  MoveL 6726 to (240.81, 149.3, 97.46) mm, rotated rx -180 ry 0 rz 180 deg; joints [-61.575, 61.202, -81.531, 63.09, 99.519, 18.047]
  Call Extruder(259.46531)
  MoveL 6727 to (240.76, 149.6, 97.46) mm, rotated rx 180 ry 0 rz 180 deg; joints [-61.639, 61.223, -81.522, 63.147, 99.485, 18.03]
  MoveL 6728 to (240.76, 149.6, 97.46) mm, rotated rx 180 ry 0 rz 180 deg; joints [-61.639, 61.223, -81.522, 63.147, 99.485, 18.03]
  Call Extruder(259.62559)
  MoveL 6729 to (240.71, 149.91, 97.46) mm, rotated rx -180 ry 0 rz -180 deg; joints [-61.702, 61.244, -81.513, 63.203, 99.453, 18.013]
  MoveL 6730 to (240.71, 149.91, 97.46) mm, rotated rx -180 ry 0 rz -180 deg; joints [-61.702, 61.244, -81.513, 63.203, 99.453, 18.013]
  Call Extruder(259.78661)
  MoveL 6731 to (240.66, 150.21, 97.46) mm, rotated rx -180 ry 0 rz -180 deg; joints [-61.765, 61.265, -81.504, 63.26, 99.419, 17.996]
  MoveL 6732 to (240.66, 150.21, 97.46) mm, rotated rx -180 ry 0 rz -180 deg; joints [-61.765, 61.265, -81.504, 63.26, 99.419, 17.996]
  Call Extruder(259.94835)
  MoveL 6733 to (240.61, 150.52, 97.46) mm, rotated rx 180 ry 0 rz 180 deg; joints [-61.828, 61.286, -81.495, 63.316, 99.387, 17.979]
  MoveL 6734 to (240.61, 150.52, 97.46) mm, rotated rx 180 ry 0 rz 180 deg; joints [-61.828, 61.286, -81.495, 63.316, 99.387, 17.979]
  Call Extruder(260.11082)
  MoveL 6735 to (240.56, 150.83, 97.46) mm, rotated rx 180 ry 0 rz 180 deg; joints [-61.891, 61.307, -81.486, 63.372, 99.354, 17.961]
  MoveL 6736 to (240.56, 150.83, 97.46) mm, rotated rx 180 ry 0 rz 180 deg; joints [-61.891, 61.307, -81.486, 63.372, 99.354, 17.961]
  Call Extruder(260.24475)
  MoveL 6737 to (240.52, 151.08, 97.46) mm, rotated rx -180 ry 0 rz 180 deg; joints [-61.944, 61.324, -81.479, 63.42, 99.327, 17.948]
  MoveL 6738 to (240.52, 151.08, 97.46) mm, rotated rx -180 ry 0 rz 180 deg; joints [-61.944, 61.324, -81.479, 63.42, 99.327, 17.948]
  Call Extruder(260.37929)
  MoveL 6739 to (240.47, 151.32, 97.46) mm, rotated rx -180 ry 0 rz 180 deg; joints [-61.998, 61.34, -81.472, 63.469, 99.299, 17.935]
  MoveL 6740 to (240.47, 151.32, 97.46) mm, rotated rx -180 ry 0 rz 180 deg; joints [-61.998, 61.34, -81.472, 63.469, 99.299, 17.935]
  Call Extruder(260.51443)
  MoveL 6741 to (240.42, 151.57, 97.46) mm, rotated rx -180 ry 0 rz 180 deg; joints [-62.052, 61.357, -81.465, 63.517, 99.272, 17.922]
  MoveL 6742 to (240.42, 151.57, 97.46) mm, rotated rx -180 ry 0 rz 180 deg; joints [-62.052, 61.357, -81.465, 63.517, 99.272, 17.922]
  Call Extruder(260.65019)
  MoveL 6743 to (240.37, 151.82, 97.46) mm, rotated rx 180 ry 0 rz -180 deg; joints [-62.105, 61.374, -81.458, 63.565, 99.245, 17.908]
  MoveL 6744 to (240.37, 151.82, 97.46) mm, rotated rx 180 ry 0 rz -180 deg; joints [-62.105, 61.374, -81.458, 63.565, 99.245, 17.908]
  Call Extruder(260.78656)
  MoveL 6745 to (240.32, 152.07, 97.46) mm, rotated rx 180 ry 0 rz -180 deg; joints [-62.159, 61.39, -81.45, 63.613, 99.218, 17.895]
  MoveL 6746 to (240.32, 152.07, 97.46) mm, rotated rx 180 ry 0 rz -180 deg; joints [-62.159, 61.39, -81.45, 63.613, 99.218, 17.895]
  Call Extruder(260.92354)
  MoveL 6747 to (240.27, 152.32, 97.46) mm, rotated rx -180 ry 0 rz 180 deg; joints [-62.212, 61.407, -81.443, 63.661, 99.191, 17.881]
  MoveL 6748 to (240.27, 152.32, 97.46) mm, rotated rx -180 ry 0 rz 180 deg; joints [-62.212, 61.407, -81.443, 63.661, 99.191, 17.881]
  Call Extruder(261.06113)
  MoveL 6749 to (240.22, 152.57, 97.46) mm, rotated rx -180 ry 0 rz 180 deg; joints [-62.265, 61.424, -81.436, 63.709, 99.164, 17.868]
  MoveL 6750 to (240.22, 152.57, 97.46) mm, rotated rx -180 ry 0 rz 180 deg; joints [-62.265, 61.424, -81.436, 63.709, 99.164, 17.868]
  Call Extruder(261.17482)
  MoveL 6751 to (240.17, 152.77, 97.46) mm, rotated rx -180 ry 0 rz 180 deg; joints [-62.31, 61.437, -81.43, 63.749, 99.142, 17.857]
  MoveL 6752 to (240.17, 152.77, 97.46) mm, rotated rx -180 ry 0 rz 180 deg; joints [-62.31, 61.437, -81.43, 63.749, 99.142, 17.857]
  Call Extruder(261.28897)
  MoveL 6753 to (240.13, 152.98, 97.46) mm, rotated rx 180 ry 0 rz 180 deg; joints [-62.355, 61.451, -81.424, 63.789, 99.119, 17.846]
  MoveL 6754 to (240.13, 152.98, 97.46) mm, rotated rx 180 ry 0 rz 180 deg; joints [-62.355, 61.451, -81.424, 63.789, 99.119, 17.846]
  Call Extruder(261.40358)
  MoveL 6755 to (240.08, 153.18, 97.46) mm, rotated rx -180 ry 0 rz 180 deg; joints [-62.399, 61.464, -81.418, 63.83, 99.097, 17.835]
  MoveL 6756 to (240.08, 153.18, 97.46) mm, rotated rx -180 ry 0 rz 180 deg; joints [-62.399, 61.464, -81.418, 63.83, 99.097, 17.835]
  Call Extruder(261.51863)
  MoveL 6757 to (240.04, 153.39, 97.46) mm, rotated rx -180 ry 0 rz 180 deg; joints [-62.444, 61.478, -81.412, 63.869, 99.075, 17.824]
  MoveL 6758 to (240.04, 153.39, 97.46) mm, rotated rx -180 ry 0 rz 180 deg; joints [-62.444, 61.478, -81.412, 63.869, 99.075, 17.824]
  Call Extruder(261.64086)
  MoveL 6759 to (239.98, 153.6, 97.46) mm, rotated rx -180 ry 0 rz -180 deg; joints [-62.493, 61.492, -81.406, 63.914, 99.051, 17.813]
  MoveL 6760 to (239.98, 153.6, 97.46) mm, rotated rx -180 ry 0 rz -180 deg; joints [-62.493, 61.492, -81.406, 63.914, 99.051, 17.813]
  Call Extruder(261.77052)
  MoveL 6761 to (239.92, 153.82, 97.46) mm, rotated rx -180 ry 0 rz 180 deg; joints [-62.547, 61.506, -81.4, 63.963, 99.026, 17.803]
  MoveL 6762 to (239.92, 153.82, 97.46) mm, rotated rx -180 ry 0 rz 180 deg; joints [-62.547, 61.506, -81.4, 63.963, 99.026, 17.803]
  Call Extruder(261.90074)
  MoveL 6763 to (239.85, 154.05, 97.46) mm, rotated rx 180 ry 0 rz 180 deg; joints [-62.601, 61.52, -81.394, 64.012, 99, 17.793]
  MoveL 6764 to (239.85, 154.05, 97.46) mm, rotated rx 180 ry 0 rz 180 deg; joints [-62.601, 61.52, -81.394, 64.012, 99, 17.793]
  Call Extruder(262.03153)
  MoveL 6765 to (239.78, 154.27, 97.46) mm, rotated rx -180 ry 0 rz -180 deg; joints [-62.654, 61.534, -81.387, 64.061, 98.975, 17.782]
  MoveL 6766 to (239.78, 154.27, 97.46) mm, rotated rx -180 ry 0 rz -180 deg; joints [-62.654, 61.534, -81.387, 64.061, 98.975, 17.782]
  Call Extruder(262.16289)
  MoveL 6767 to (239.71, 154.49, 97.46) mm, rotated rx -180 ry 0 rz 180 deg; joints [-62.708, 61.548, -81.381, 64.11, 98.95, 17.772]
  MoveL 6768 to (239.71, 154.49, 97.46) mm, rotated rx -180 ry 0 rz 180 deg; joints [-62.708, 61.548, -81.381, 64.11, 98.95, 17.772]
  Call Extruder(262.27479)
  MoveL 6769 to (239.65, 154.68, 97.46) mm, rotated rx -180 ry 0 rz 180 deg; joints [-62.754, 61.56, -81.376, 64.152, 98.928, 17.763]
  MoveL 6770 to (239.65, 154.68, 97.46) mm, rotated rx -180 ry 0 rz 180 deg; joints [-62.754, 61.56, -81.376, 64.152, 98.928, 17.763]
  Call Extruder(262.38714)
  MoveL 6771 to (239.59, 154.87, 97.46) mm, rotated rx -180 ry 0 rz 180 deg; joints [-62.801, 61.572, -81.371, 64.195, 98.907, 17.754]
  MoveL 6772 to (239.59, 154.87, 97.46) mm, rotated rx -180 ry 0 rz 180 deg; joints [-62.801, 61.572, -81.371, 64.195, 98.907, 17.754]
  Call Extruder(262.49993)
  MoveL 6773 to (239.53, 155.06, 97.46) mm, rotated rx -180 ry 0 rz 180 deg; joints [-62.847, 61.584, -81.365, 64.237, 98.885, 17.746]
  MoveL 6774 to (239.53, 155.06, 97.46) mm, rotated rx -180 ry 0 rz 180 deg; joints [-62.847, 61.584, -81.365, 64.237, 98.885, 17.746]
  Call Extruder(262.61316)
  MoveL 6775 to (239.47, 155.25, 97.46) mm, rotated rx -180 ry 0 rz 180 deg; joints [-62.893, 61.595, -81.36, 64.279, 98.864, 17.737]
  MoveL 6776 to (239.47, 155.25, 97.46) mm, rotated rx -180 ry 0 rz 180 deg; joints [-62.893, 61.595, -81.36, 64.279, 98.864, 17.737]
  Call Extruder(262.72684)
  MoveL 6777 to (239.41, 155.44, 97.46) mm, rotated rx 180 ry 0 rz -180 deg; joints [-62.939, 61.607, -81.355, 64.321, 98.842, 17.729]
  MoveL 6778 to (239.41, 155.44, 97.46) mm, rotated rx 180 ry 0 rz -180 deg; joints [-62.939, 61.607, -81.355, 64.321, 98.842, 17.729]
  Call Extruder(262.90880)
  MoveL 6779 to (239.29, 155.73, 97.46) mm, rotated rx 180 ry 0 rz 180 deg; joints [-63.018, 61.624, -81.347, 64.393, 98.807, 17.717]
  MoveL 6780 to (239.29, 155.73, 97.46) mm, rotated rx 180 ry 0 rz 180 deg; joints [-63.018, 61.624, -81.347, 64.393, 98.807, 17.717]
  Call Extruder(263.09151)
  MoveL 6781 to (239.17, 156.02, 97.46) mm, rotated rx 180 ry 0 rz 180 deg; joints [-63.097, 61.642, -81.339, 64.466, 98.773, 17.706]
  MoveL 6782 to (239.17, 156.02, 97.46) mm, rotated rx 180 ry 0 rz 180 deg; joints [-63.097, 61.642, -81.339, 64.466, 98.773, 17.706]
  Call Extruder(263.26194)
  MoveL 6783 to (239.05, 156.29, 97.46) mm, rotated rx 180 ry 0 rz -180 deg; joints [-63.17, 61.657, -81.332, 64.533, 98.74, 17.696]
  MoveL 6784 to (239.05, 156.29, 97.46) mm, rotated rx 180 ry 0 rz -180 deg; joints [-63.17, 61.657, -81.332, 64.533, 98.74, 17.696]
  Call Extruder(263.41995)
  MoveL 6785 to (238.94, 156.54, 97.46) mm, rotated rx -180 ry 0 rz -180 deg; joints [-63.238, 61.672, -81.325, 64.596, 98.711, 17.686]
  MoveL 6786 to (238.94, 156.54, 97.46) mm, rotated rx -180 ry 0 rz -180 deg; joints [-63.238, 61.672, -81.325, 64.596, 98.711, 17.686]
  Call Extruder(263.57856)
  MoveL 6787 to (238.84, 156.79, 97.46) mm, rotated rx -180 ry 0 rz -180 deg; joints [-63.306, 61.687, -81.319, 64.658, 98.681, 17.677]
  MoveL 6788 to (238.84, 156.79, 97.46) mm, rotated rx -180 ry 0 rz -180 deg; joints [-63.306, 61.687, -81.319, 64.658, 98.681, 17.677]
  Call Extruder(263.78473)
  MoveL 6789 to (238.66, 157.09, 97.46) mm, rotated rx -180 ry 0 rz 180 deg; joints [-63.401, 61.703, -81.311, 64.747, 98.642, 17.669]
  MoveL 6790 to (238.66, 157.09, 97.46) mm, rotated rx -180 ry 0 rz 180 deg; joints [-63.401, 61.703, -81.311, 64.747, 98.642, 17.669]
  Call Extruder(263.99168)
  MoveL 6791 to (238.49, 157.4, 97.46) mm, rotated rx 180 ry 0 rz 180 deg; joints [-63.497, 61.719, -81.304, 64.836, 98.603, 17.661]
  MoveL 6792 to (238.49, 157.4, 97.46) mm, rotated rx 180 ry 0 rz 180 deg; joints [-63.497, 61.719, -81.304, 64.836, 98.603, 17.661]
  Call Extruder(264.19941)
  MoveL 6793 to (238.31, 157.7, 97.46) mm, rotated rx 180 ry 0 rz 180 deg; joints [-63.592, 61.735, -81.297, 64.924, 98.564, 17.653]
  MoveL 6794 to (238.31, 157.7, 97.46) mm, rotated rx 180 ry 0 rz 180 deg; joints [-63.592, 61.735, -81.297, 64.924, 98.564, 17.653]
  Call Extruder(264.40791)
  MoveL 6795 to (238.13, 158.01, 97.46) mm, rotated rx 180 ry 0 rz 180 deg; joints [-63.687, 61.752, -81.289, 65.013, 98.525, 17.645]
  MoveL 6796 to (238.13, 158.01, 97.46) mm, rotated rx 180 ry 0 rz 180 deg; joints [-63.687, 61.752, -81.289, 65.013, 98.525, 17.645]
  Call Extruder(264.58745)
  MoveL 6797 to (237.96, 158.25, 97.46) mm, rotated rx 180 ry 0 rz 180 deg; joints [-63.774, 61.763, -81.284, 65.094, 98.491, 17.642]
  MoveL 6798 to (237.96, 158.25, 97.46) mm, rotated rx 180 ry 0 rz 180 deg; joints [-63.774, 61.763, -81.284, 65.094, 98.491, 17.642]
  Call Extruder(264.92086)
  MoveL 6799 to (237.63, 158.7, 97.46) mm, rotated rx -180 ry 0 rz -180 deg; joints [-63.934, 61.785, -81.274, 65.244, 98.43, 17.635]
  MoveL 6800 to (237.63, 158.7, 97.46) mm, rotated rx -180 ry 0 rz -180 deg; joints [-63.934, 61.785, -81.274, 65.244, 98.43, 17.635]
  Call Extruder(265.25545)
  MoveL 6801 to (237.3, 159.15, 97.46) mm, rotated rx 180 ry 0 rz 180 deg; joints [-64.094, 61.807, -81.263, 65.393, 98.368, 17.628]
  Call Extruder(266.08341)
  MoveL 6802 to (236.39, 160.19, 97.46) mm, rotated rx -180 ry 0 rz -180 deg; joints [-64.505, 61.852, -81.243, 65.781, 98.216, 17.625]
  Call Extruder(266.91134)
  MoveL 6803 to (235.35, 161.1, 97.46) mm, rotated rx 180 ry 0 rz -180 deg; joints [-64.933, 61.884, -81.228, 66.187, 98.068, 17.64]
  Call Extruder(267.07865)
  MoveL 6804 to (235.13, 161.27, 97.46) mm, rotated rx -180 ry 0 rz 180 deg; joints [-65.021, 61.888, -81.226, 66.271, 98.038, 17.646]
  MoveL 6805 to (235.13, 161.27, 97.46) mm, rotated rx -180 ry 0 rz 180 deg; joints [-65.021, 61.888, -81.226, 66.271, 98.038, 17.646]
  Call Extruder(267.41207)
  MoveL 6806 to (234.68, 161.6, 97.46) mm, rotated rx 180 ry 0 rz 180 deg; joints [-65.197, 61.897, -81.221, 66.439, 97.98, 17.658]
  MoveL 6807 to (234.68, 161.6, 97.46) mm, rotated rx 180 ry 0 rz 180 deg; joints [-65.197, 61.897, -81.221, 66.439, 97.98, 17.658]
  Call Extruder(267.74432)
  MoveL 6808 to (234.23, 161.92, 97.46) mm, rotated rx -180 ry 0 rz 180 deg; joints [-65.374, 61.906, -81.217, 66.607, 97.921, 17.669]
  MoveL 6809 to (234.23, 161.92, 97.46) mm, rotated rx -180 ry 0 rz 180 deg; joints [-65.374, 61.906, -81.217, 66.607, 97.921, 17.669]
  Call Extruder(267.86197)
  MoveL 6810 to (234.05, 162.02, 97.46) mm, rotated rx 180 ry 0 rz -180 deg; joints [-65.437, 61.908, -81.216, 66.667, 97.901, 17.675]
  MoveL 6811 to (234.05, 162.02, 97.46) mm, rotated rx 180 ry 0 rz -180 deg; joints [-65.437, 61.908, -81.216, 66.667, 97.901, 17.675]
  Call Extruder(268.06970)
  MoveL 6812 to (233.75, 162.2, 97.46) mm, rotated rx -180 ry 0 rz 180 deg; joints [-65.549, 61.91, -81.215, 66.775, 97.865, 17.686]
  MoveL 6813 to (233.75, 162.2, 97.46) mm, rotated rx -180 ry 0 rz 180 deg; joints [-65.549, 61.91, -81.215, 66.775, 97.865, 17.686]
  Call Extruder(268.27665)
  MoveL 6814 to (233.45, 162.37, 97.46) mm, rotated rx -180 ry 0 rz 180 deg; joints [-65.662, 61.913, -81.214, 66.882, 97.829, 17.697]
  MoveL 6815 to (233.45, 162.37, 97.46) mm, rotated rx -180 ry 0 rz 180 deg; joints [-65.662, 61.913, -81.214, 66.882, 97.829, 17.697]
  Call Extruder(268.48282)
  MoveL 6816 to (233.14, 162.55, 97.46) mm, rotated rx 180 ry 0 rz 180 deg; joints [-65.774, 61.916, -81.212, 66.99, 97.793, 17.708]
  MoveL 6817 to (233.14, 162.55, 97.46) mm, rotated rx 180 ry 0 rz 180 deg; joints [-65.774, 61.916, -81.212, 66.99, 97.793, 17.708]
  Call Extruder(268.66449)
  MoveL 6818 to (232.87, 162.69, 97.46) mm, rotated rx 180 ry 0 rz 180 deg; joints [-65.874, 61.917, -81.212, 67.085, 97.762, 17.719]
  MoveL 6819 to (232.87, 162.69, 97.46) mm, rotated rx 180 ry 0 rz 180 deg; joints [-65.874, 61.917, -81.212, 67.085, 97.762, 17.719]
  Call Extruder(268.82246)
  MoveL 6820 to (232.62, 162.8, 97.46) mm, rotated rx 180 ry 0 rz 180 deg; joints [-65.961, 61.917, -81.212, 67.169, 97.736, 17.731]
  MoveL 6821 to (232.62, 162.8, 97.46) mm, rotated rx 180 ry 0 rz 180 deg; joints [-65.961, 61.917, -81.212, 67.169, 97.736, 17.731]
  Call Extruder(268.97983)
  MoveL 6822 to (232.37, 162.9, 97.46) mm, rotated rx -180 ry 0 rz 180 deg; joints [-66.048, 61.917, -81.212, 67.253, 97.709, 17.742]
  MoveL 6823 to (232.37, 162.9, 97.46) mm, rotated rx -180 ry 0 rz 180 deg; joints [-66.048, 61.917, -81.212, 67.253, 97.709, 17.742]
  Call Extruder(269.16257)
  MoveL 6824 to (232.07, 163.03, 97.46) mm, rotated rx 180 ry 0 rz -180 deg; joints [-66.149, 61.916, -81.212, 67.351, 97.679, 17.756]
  MoveL 6825 to (232.07, 163.03, 97.46) mm, rotated rx 180 ry 0 rz -180 deg; joints [-66.149, 61.916, -81.212, 67.351, 97.679, 17.756]
  Call Extruder(269.34456)
  MoveL 6826 to (231.78, 163.15, 97.46) mm, rotated rx -180 ry 0 rz 180 deg; joints [-66.251, 61.916, -81.213, 67.448, 97.648, 17.77]
  MoveL 6827 to (231.78, 163.15, 97.46) mm, rotated rx -180 ry 0 rz 180 deg; joints [-66.251, 61.916, -81.213, 67.448, 97.648, 17.77]
  Call Extruder(269.49190)
  MoveL 6828 to (231.54, 163.24, 97.46) mm, rotated rx 180 ry 0 rz -180 deg; joints [-66.333, 61.914, -81.213, 67.528, 97.624, 17.782]
  MoveL 6829 to (231.54, 163.24, 97.46) mm, rotated rx 180 ry 0 rz -180 deg; joints [-66.333, 61.914, -81.213, 67.528, 97.624, 17.782]
  Call Extruder(269.60512)
  MoveL 6830 to (231.35, 163.3, 97.46) mm, rotated rx -180 ry 0 rz -180 deg; joints [-66.397, 61.913, -81.214, 67.589, 97.605, 17.792]
  MoveL 6831 to (231.35, 163.3, 97.46) mm, rotated rx -180 ry 0 rz -180 deg; joints [-66.397, 61.913, -81.214, 67.589, 97.605, 17.792]
  Call Extruder(269.71789)
  MoveL 6832 to (231.17, 163.36, 97.46) mm, rotated rx 180 ry 0 rz 180 deg; joints [-66.46, 61.911, -81.215, 67.65, 97.587, 17.803]
  MoveL 6833 to (231.17, 163.36, 97.46) mm, rotated rx 180 ry 0 rz 180 deg; joints [-66.46, 61.911, -81.215, 67.65, 97.587, 17.803]
  Call Extruder(269.83022)
  MoveL 6834 to (230.98, 163.42, 97.46) mm, rotated rx -180 ry 0 rz 180 deg; joints [-66.524, 61.91, -81.215, 67.711, 97.568, 17.813]
  MoveL 6835 to (230.98, 163.42, 97.46) mm, rotated rx -180 ry 0 rz 180 deg; joints [-66.524, 61.91, -81.215, 67.711, 97.568, 17.813]
  Call Extruder(269.94211)
  MoveL 6836 to (230.79, 163.48, 97.46) mm, rotated rx 180 ry 0 rz 180 deg; joints [-66.587, 61.908, -81.216, 67.772, 97.55, 17.823]
  MoveL 6837 to (230.79, 163.48, 97.46) mm, rotated rx 180 ry 0 rz 180 deg; joints [-66.587, 61.908, -81.216, 67.772, 97.55, 17.823]
  Call Extruder(270.06351)
  MoveL 6838 to (230.58, 163.55, 97.46) mm, rotated rx -180 ry 0 rz -180 deg; joints [-66.656, 61.906, -81.217, 67.839, 97.529, 17.834]
  MoveL 6839 to (230.58, 163.55, 97.46) mm, rotated rx -180 ry 0 rz -180 deg; joints [-66.656, 61.906, -81.217, 67.839, 97.529, 17.834]
  Call Extruder(270.19433)
  MoveL 6840 to (230.36, 163.62, 97.46) mm, rotated rx -180 ry 0 rz -180 deg; joints [-66.731, 61.904, -81.218, 67.911, 97.508, 17.847]
  MoveL 6841 to (230.36, 163.62, 97.46) mm, rotated rx -180 ry 0 rz -180 deg; joints [-66.731, 61.904, -81.218, 67.911, 97.508, 17.847]
  Call Extruder(270.32458)
  MoveL 6842 to (230.14, 163.68, 97.46) mm, rotated rx 180 ry 0 rz -180 deg; joints [-66.805, 61.902, -81.219, 67.983, 97.486, 17.859]
  MoveL 6843 to (230.14, 163.68, 97.46) mm, rotated rx 180 ry 0 rz -180 deg; joints [-66.805, 61.902, -81.219, 67.983, 97.486, 17.859]
  Call Extruder(270.45426)
  MoveL 6844 to (229.91, 163.75, 97.46) mm, rotated rx 180 ry 0 rz -180 deg; joints [-66.88, 61.9, -81.22, 68.056, 97.464, 17.871]
  MoveL 6845 to (229.91, 163.75, 97.46) mm, rotated rx 180 ry 0 rz -180 deg; joints [-66.88, 61.9, -81.22, 68.056, 97.464, 17.871]
  Call Extruder(270.58338)
  MoveL 6846 to (229.69, 163.82, 97.46) mm, rotated rx 180 ry 0 rz 180 deg; joints [-66.955, 61.898, -81.221, 68.128, 97.443, 17.884]
  MoveL 6847 to (229.69, 163.82, 97.46) mm, rotated rx 180 ry 0 rz 180 deg; joints [-66.955, 61.898, -81.221, 68.128, 97.443, 17.884]
  Call Extruder(270.69845)
  MoveL 6848 to (229.48, 163.86, 97.46) mm, rotated rx -180 ry 0 rz 180 deg; joints [-67.021, 61.894, -81.223, 68.192, 97.424, 17.896]
  MoveL 6849 to (229.48, 163.86, 97.46) mm, rotated rx -180 ry 0 rz 180 deg; joints [-67.021, 61.894, -81.223, 68.192, 97.424, 17.896]
  Call Extruder(270.81308)
  MoveL 6850 to (229.28, 163.91, 97.46) mm, rotated rx -180 ry 0 rz 180 deg; joints [-67.087, 61.891, -81.224, 68.256, 97.405, 17.909]
  MoveL 6851 to (229.28, 163.91, 97.46) mm, rotated rx -180 ry 0 rz 180 deg; joints [-67.087, 61.891, -81.224, 68.256, 97.405, 17.909]
  Call Extruder(270.92725)
  MoveL 6852 to (229.08, 163.95, 97.46) mm, rotated rx 180 ry 0 rz -180 deg; joints [-67.153, 61.888, -81.226, 68.32, 97.387, 17.921]
  MoveL 6853 to (229.08, 163.95, 97.46) mm, rotated rx 180 ry 0 rz -180 deg; joints [-67.153, 61.888, -81.226, 68.32, 97.387, 17.921]
  Call Extruder(271.04096)
  MoveL 6854 to (228.87, 164, 97.46) mm, rotated rx -180 ry 0 rz 180 deg; joints [-67.22, 61.885, -81.227, 68.384, 97.368, 17.934]
  MoveL 6855 to (228.87, 164, 97.46) mm, rotated rx -180 ry 0 rz 180 deg; joints [-67.22, 61.885, -81.227, 68.384, 97.368, 17.934]
  Call Extruder(271.16638)
  MoveL 6856 to (228.65, 164.04, 97.46) mm, rotated rx -180 ry 0 rz -180 deg; joints [-67.293, 61.881, -81.229, 68.455, 97.348, 17.948]
  MoveL 6857 to (228.65, 164.04, 97.46) mm, rotated rx -180 ry 0 rz -180 deg; joints [-67.293, 61.881, -81.229, 68.455, 97.348, 17.948]
  Call Extruder(271.30336)
  MoveL 6858 to (228.4, 164.09, 97.46) mm, rotated rx 180 ry 0 rz -180 deg; joints [-67.373, 61.877, -81.231, 68.532, 97.325, 17.963]
  MoveL 6859 to (228.4, 164.09, 97.46) mm, rotated rx 180 ry 0 rz -180 deg; joints [-67.373, 61.877, -81.231, 68.532, 97.325, 17.963]
  Call Extruder(271.43973)
  MoveL 6860 to (228.15, 164.14, 97.46) mm, rotated rx -180 ry 0 rz 180 deg; joints [-67.453, 61.873, -81.233, 68.61, 97.303, 17.979]
  MoveL 6861 to (228.15, 164.14, 97.46) mm, rotated rx -180 ry 0 rz 180 deg; joints [-67.453, 61.873, -81.233, 68.61, 97.303, 17.979]
  Call Extruder(271.57549)
  MoveL 6862 to (227.9, 164.19, 97.46) mm, rotated rx 180 ry 0 rz -180 deg; joints [-67.534, 61.869, -81.235, 68.688, 97.28, 17.994]
  MoveL 6863 to (227.9, 164.19, 97.46) mm, rotated rx 180 ry 0 rz -180 deg; joints [-67.534, 61.869, -81.235, 68.688, 97.28, 17.994]
  Call Extruder(271.71064)
  MoveL 6864 to (227.65, 164.24, 97.46) mm, rotated rx -180 ry 0 rz -180 deg; joints [-67.614, 61.865, -81.237, 68.766, 97.257, 18.01]
  MoveL 6865 to (227.65, 164.24, 97.46) mm, rotated rx -180 ry 0 rz -180 deg; joints [-67.614, 61.865, -81.237, 68.766, 97.257, 18.01]
  Call Extruder(271.84517)
  MoveL 6866 to (227.4, 164.29, 97.46) mm, rotated rx 180 ry 0 rz -180 deg; joints [-67.695, 61.861, -81.238, 68.843, 97.235, 18.025]
  MoveL 6867 to (227.4, 164.29, 97.46) mm, rotated rx 180 ry 0 rz -180 deg; joints [-67.695, 61.861, -81.238, 68.843, 97.235, 18.025]
  Call Extruder(271.97910)
  MoveL 6868 to (227.15, 164.34, 97.46) mm, rotated rx -180 ry 0 rz -180 deg; joints [-67.775, 61.857, -81.24, 68.921, 97.212, 18.04]
  MoveL 6869 to (227.15, 164.34, 97.46) mm, rotated rx -180 ry 0 rz -180 deg; joints [-67.775, 61.857, -81.24, 68.921, 97.212, 18.04]
  Call Extruder(272.12696)
  MoveL 6870 to (226.87, 164.39, 97.46) mm, rotated rx 180 ry 0 rz 180 deg; joints [-67.864, 61.852, -81.243, 69.007, 97.187, 18.058]
  MoveL 6871 to (226.87, 164.39, 97.46) mm, rotated rx 180 ry 0 rz 180 deg; joints [-67.864, 61.852, -81.243, 69.007, 97.187, 18.058]
  Call Extruder(272.28870)
  MoveL 6872 to (226.57, 164.44, 97.46) mm, rotated rx 180 ry 0 rz 180 deg; joints [-67.961, 61.846, -81.245, 69.102, 97.16, 18.078]
  MoveL 6873 to (226.57, 164.44, 97.46) mm, rotated rx 180 ry 0 rz 180 deg; joints [-67.961, 61.846, -81.245, 69.102, 97.16, 18.078]
  Call Extruder(272.44972)
  MoveL 6874 to (226.26, 164.49, 97.46) mm, rotated rx 180 ry 0 rz 180 deg; joints [-68.059, 61.84, -81.248, 69.196, 97.133, 18.097]
  MoveL 6875 to (226.26, 164.49, 97.46) mm, rotated rx 180 ry 0 rz 180 deg; joints [-68.059, 61.84, -81.248, 69.196, 97.133, 18.097]
  Call Extruder(272.61000)
  MoveL 6876 to (225.96, 164.53, 97.46) mm, rotated rx -180 ry 0 rz 180 deg; joints [-68.156, 61.834, -81.251, 69.29, 97.105, 18.117]
  MoveL 6877 to (225.96, 164.53, 97.46) mm, rotated rx -180 ry 0 rz 180 deg; joints [-68.156, 61.834, -81.251, 69.29, 97.105, 18.117]
  Call Extruder(272.76956)
  MoveL 6878 to (225.65, 164.58, 97.46) mm, rotated rx -180 ry 0 rz 180 deg; joints [-68.254, 61.829, -81.253, 69.385, 97.078, 18.136]
  MoveL 6879 to (225.65, 164.58, 97.46) mm, rotated rx -180 ry 0 rz 180 deg; joints [-68.254, 61.829, -81.253, 69.385, 97.078, 18.136]
  Call Extruder(272.92838)
  MoveL 6880 to (225.34, 164.63, 97.46) mm, rotated rx -180 ry 0 rz -180 deg; joints [-68.351, 61.823, -81.256, 69.479, 97.05, 18.155]
  MoveL 6881 to (225.34, 164.63, 97.46) mm, rotated rx -180 ry 0 rz -180 deg; joints [-68.351, 61.823, -81.256, 69.479, 97.05, 18.155]
  Call Extruder(273.10706)
  MoveL 6882 to (225, 164.68, 97.46) mm, rotated rx 180 ry 0 rz -180 deg; joints [-68.461, 61.816, -81.259, 69.586, 97.02, 18.178]
  MoveL 6883 to (225, 164.68, 97.46) mm, rotated rx 180 ry 0 rz -180 deg; joints [-68.461, 61.816, -81.259, 69.586, 97.02, 18.178]
  Call Extruder(273.30550)
  MoveL 6884 to (224.61, 164.73, 97.46) mm, rotated rx 180 ry 0 rz -180 deg; joints [-68.583, 61.808, -81.263, 69.704, 96.986, 18.204]
  MoveL 6885 to (224.61, 164.73, 97.46) mm, rotated rx 180 ry 0 rz -180 deg; joints [-68.583, 61.808, -81.263, 69.704, 96.986, 18.204]
  Call Extruder(273.50307)
  MoveL 6886 to (224.22, 164.77, 97.46) mm, rotated rx -180 ry 0 rz 180 deg; joints [-68.706, 61.799, -81.267, 69.822, 96.952, 18.229]
  MoveL 6887 to (224.22, 164.77, 97.46) mm, rotated rx -180 ry 0 rz 180 deg; joints [-68.706, 61.799, -81.267, 69.822, 96.952, 18.229]
  Call Extruder(273.69978)
  MoveL 6888 to (223.84, 164.82, 97.46) mm, rotated rx -180 ry 0 rz 180 deg; joints [-68.828, 61.791, -81.271, 69.941, 96.917, 18.255]
  MoveL 6889 to (223.84, 164.82, 97.46) mm, rotated rx -180 ry 0 rz 180 deg; joints [-68.828, 61.791, -81.271, 69.941, 96.917, 18.255]
  Call Extruder(273.89562)
  MoveL 6890 to (223.45, 164.86, 97.46) mm, rotated rx -180 ry 0 rz 180 deg; joints [-68.951, 61.783, -81.274, 70.06, 96.883, 18.28]
  MoveL 6891 to (223.45, 164.86, 97.46) mm, rotated rx -180 ry 0 rz 180 deg; joints [-68.951, 61.783, -81.274, 70.06, 96.883, 18.28]
  Call Extruder(274.19098)
  MoveL 6892 to (222.86, 164.91, 97.46) mm, rotated rx 180 ry 0 rz 180 deg; joints [-69.135, 61.769, -81.281, 70.238, 96.832, 18.32]
  MoveL 6893 to (222.86, 164.91, 97.46) mm, rotated rx 180 ry 0 rz 180 deg; joints [-69.135, 61.769, -81.281, 70.238, 96.832, 18.32]
  Call Extruder(274.48500)
  MoveL 6894 to (222.27, 164.96, 97.46) mm, rotated rx 180 ry 0 rz 180 deg; joints [-69.319, 61.755, -81.287, 70.416, 96.781, 18.36]
  MoveL 6895 to (222.27, 164.96, 97.46) mm, rotated rx 180 ry 0 rz 180 deg; joints [-69.319, 61.755, -81.287, 70.416, 96.781, 18.36]
  Call Extruder(274.77770)
  MoveL 6896 to (221.68, 165, 97.46) mm, rotated rx -180 ry 0 rz 180 deg; joints [-69.504, 61.742, -81.294, 70.595, 96.729, 18.4]
  MoveL 6897 to (221.68, 165, 97.46) mm, rotated rx -180 ry 0 rz 180 deg; joints [-69.504, 61.742, -81.294, 70.595, 96.729, 18.4]
  Call Extruder(275.35114)
  MoveL 6898 to (220.52, 165.05, 97.46) mm, rotated rx 180 ry 0 rz 180 deg; joints [-69.864, 61.712, -81.307, 70.944, 96.63, 18.482]
  MoveL 6899 to (220.52, 165.05, 97.46) mm, rotated rx 180 ry 0 rz 180 deg; joints [-69.864, 61.712, -81.307, 70.944, 96.63, 18.482]
  Call Extruder(276.06515)
  MoveL 6900 to (219.06, 165.09, 97.46) mm, rotated rx 180 ry 0 rz 180 deg; joints [-70.315, 61.673, -81.325, 71.38, 96.505, 18.584]
  Call Extruder(392.91189)
  MoveL 6901 to (-19.06, 165.09, 97.46) mm, rotated rx -180 ry 0 rz 180 deg; joints [-137.325, 66.695, -77.852, 136.78, 81.821, 7.615]
  Call Extruder(393.34049)
  MoveL 6902 to (-19.94, 165.07, 97.46) mm, rotated rx -180 ry 0 rz -180 deg; joints [-137.467, 66.734, -77.812, 136.93, 81.861, 7.539]
  MoveL 6903 to (-19.94, 165.07, 97.46) mm, rotated rx -180 ry 0 rz -180 deg; joints [-137.467, 66.734, -77.812, 136.93, 81.861, 7.539]
  Call Extruder(393.91395)
  MoveL 6904 to (-21.1, 165.03, 97.46) mm, rotated rx 180 ry 0 rz -180 deg; joints [-137.659, 66.786, -77.758, 137.132, 81.913, 7.44]
  MoveL 6905 to (-21.1, 165.03, 97.46) mm, rotated rx 180 ry 0 rz -180 deg; joints [-137.659, 66.786, -77.758, 137.132, 81.913, 7.44]
  Call Extruder(394.34824)
  MoveL 6906 to (-21.97, 164.98, 97.46) mm, rotated rx -180 ry 0 rz 180 deg; joints [-137.804, 66.825, -77.719, 137.285, 81.951, 7.366]
  MoveL 6907 to (-21.97, 164.98, 97.46) mm, rotated rx -180 ry 0 rz 180 deg; joints [-137.804, 66.825, -77.719, 137.285, 81.951, 7.366]
  Call Extruder(394.64227)
  MoveL 6908 to (-22.56, 164.93, 97.46) mm, rotated rx 180 ry 0 rz 180 deg; joints [-137.905, 66.85, -77.692, 137.391, 81.976, 7.316]
  MoveL 6909 to (-22.56, 164.93, 97.46) mm, rotated rx 180 ry 0 rz 180 deg; joints [-137.905, 66.85, -77.692, 137.391, 81.976, 7.316]
  Call Extruder(394.93763)
  MoveL 6910 to (-23.15, 164.89, 97.46) mm, rotated rx 180 ry 0 rz 180 deg; joints [-138.004, 66.875, -77.666, 137.496, 82.002, 7.267]
  MoveL 6911 to (-23.15, 164.89, 97.46) mm, rotated rx 180 ry 0 rz 180 deg; joints [-138.004, 66.875, -77.666, 137.496, 82.002, 7.267]
  Call Extruder(395.18385)
  MoveL 6912 to (-23.64, 164.84, 97.46) mm, rotated rx -180 ry 0 rz -180 deg; joints [-138.088, 66.896, -77.645, 137.584, 82.022, 7.227]
  MoveL 6913 to (-23.64, 164.84, 97.46) mm, rotated rx -180 ry 0 rz -180 deg; joints [-138.088, 66.896, -77.645, 137.584, 82.022, 7.227]
  Call Extruder(395.38056)
  MoveL 6914 to (-24.03, 164.79, 97.46) mm, rotated rx 180 ry 0 rz 180 deg; joints [-138.156, 66.912, -77.628, 137.655, 82.038, 7.195]
  MoveL 6915 to (-24.03, 164.79, 97.46) mm, rotated rx 180 ry 0 rz 180 deg; joints [-138.156, 66.912, -77.628, 137.655, 82.038, 7.195]
  Call Extruder(395.57813)
  MoveL 6916 to (-24.42, 164.75, 97.46) mm, rotated rx 180 ry 0 rz -180 deg; joints [-138.224, 66.928, -77.611, 137.726, 82.054, 7.163]
  MoveL 6917 to (-24.42, 164.75, 97.46) mm, rotated rx 180 ry 0 rz -180 deg; joints [-138.224, 66.928, -77.611, 137.726, 82.054, 7.163]
  Call Extruder(395.77657)
  MoveL 6918 to (-24.8, 164.7, 97.46) mm, rotated rx 180 ry 0 rz 180 deg; joints [-138.292, 66.944, -77.594, 137.797, 82.07, 7.132]
  MoveL 6919 to (-24.8, 164.7, 97.46) mm, rotated rx 180 ry 0 rz 180 deg; joints [-138.292, 66.944, -77.594, 137.797, 82.07, 7.132]
  Call Extruder(395.97588)
  MoveL 6920 to (-25.19, 164.66, 97.46) mm, rotated rx -180 ry 0 rz 180 deg; joints [-138.359, 66.96, -77.577, 137.867, 82.086, 7.1]
  MoveL 6921 to (-25.19, 164.66, 97.46) mm, rotated rx -180 ry 0 rz 180 deg; joints [-138.359, 66.96, -77.577, 137.867, 82.086, 7.1]
  Call Extruder(396.13471)
  MoveL 6922 to (-25.5, 164.61, 97.46) mm, rotated rx -180 ry 0 rz 180 deg; joints [-138.415, 66.972, -77.564, 137.925, 82.097, 7.075]
  MoveL 6923 to (-25.5, 164.61, 97.46) mm, rotated rx -180 ry 0 rz 180 deg; joints [-138.415, 66.972, -77.564, 137.925, 82.097, 7.075]
  Call Extruder(396.29427)
  MoveL 6924 to (-25.8, 164.56, 97.46) mm, rotated rx 180 ry 0 rz 180 deg; joints [-138.47, 66.984, -77.551, 137.983, 82.109, 7.051]
  MoveL 6925 to (-25.8, 164.56, 97.46) mm, rotated rx 180 ry 0 rz 180 deg; joints [-138.47, 66.984, -77.551, 137.983, 82.109, 7.051]
  Call Extruder(396.45456)
  MoveL 6926 to (-26.11, 164.51, 97.46) mm, rotated rx -180 ry 0 rz 180 deg; joints [-138.525, 66.996, -77.539, 138.04, 82.121, 7.027]
  MoveL 6927 to (-26.11, 164.51, 97.46) mm, rotated rx -180 ry 0 rz 180 deg; joints [-138.525, 66.996, -77.539, 138.04, 82.121, 7.027]
  Call Extruder(396.61557)
  MoveL 6928 to (-26.41, 164.46, 97.46) mm, rotated rx 180 ry 0 rz 180 deg; joints [-138.58, 67.008, -77.526, 138.098, 82.133, 7.002]
  MoveL 6929 to (-26.41, 164.46, 97.46) mm, rotated rx 180 ry 0 rz 180 deg; joints [-138.58, 67.008, -77.526, 138.098, 82.133, 7.002]
  Call Extruder(396.77732)
  MoveL 6930 to (-26.72, 164.41, 97.46) mm, rotated rx 180 ry 0 rz 180 deg; joints [-138.635, 67.021, -77.513, 138.155, 82.145, 6.978]
  MoveL 6931 to (-26.72, 164.41, 97.46) mm, rotated rx 180 ry 0 rz 180 deg; joints [-138.635, 67.021, -77.513, 138.155, 82.145, 6.978]
  Call Extruder(396.93979)
  MoveL 6932 to (-27.02, 164.36, 97.46) mm, rotated rx 180 ry 0 rz 180 deg; joints [-138.69, 67.033, -77.5, 138.212, 82.157, 6.953]
  MoveL 6933 to (-27.02, 164.36, 97.46) mm, rotated rx 180 ry 0 rz 180 deg; joints [-138.69, 67.033, -77.5, 138.212, 82.157, 6.953]
  Call Extruder(397.07371)
  MoveL 6934 to (-27.28, 164.32, 97.46) mm, rotated rx 180 ry 0 rz 180 deg; joints [-138.736, 67.042, -77.489, 138.261, 82.166, 6.934]
  MoveL 6935 to (-27.28, 164.32, 97.46) mm, rotated rx 180 ry 0 rz 180 deg; joints [-138.736, 67.042, -77.489, 138.261, 82.166, 6.934]
  Call Extruder(397.20825)
  MoveL 6936 to (-27.52, 164.27, 97.46) mm, rotated rx -180 ry 0 rz 180 deg; joints [-138.783, 67.052, -77.479, 138.309, 82.175, 6.914]
  MoveL 6937 to (-27.52, 164.27, 97.46) mm, rotated rx -180 ry 0 rz 180 deg; joints [-138.783, 67.052, -77.479, 138.309, 82.175, 6.914]
  Call Extruder(397.34340)
  MoveL 6938 to (-27.77, 164.22, 97.46) mm, rotated rx -180 ry 0 rz 180 deg; joints [-138.829, 67.061, -77.469, 138.357, 82.184, 6.895]
  MoveL 6939 to (-27.77, 164.22, 97.46) mm, rotated rx -180 ry 0 rz 180 deg; joints [-138.829, 67.061, -77.469, 138.357, 82.184, 6.895]
  Call Extruder(397.47915)
  MoveL 6940 to (-28.02, 164.17, 97.46) mm, rotated rx -180 ry 0 rz 180 deg; joints [-138.875, 67.071, -77.459, 138.405, 82.193, 6.875]
  MoveL 6941 to (-28.02, 164.17, 97.46) mm, rotated rx -180 ry 0 rz 180 deg; joints [-138.875, 67.071, -77.459, 138.405, 82.193, 6.875]
  Call Extruder(397.61552)
  MoveL 6942 to (-28.27, 164.12, 97.46) mm, rotated rx -180 ry 0 rz 180 deg; joints [-138.921, 67.08, -77.449, 138.453, 82.203, 6.856]
  MoveL 6943 to (-28.27, 164.12, 97.46) mm, rotated rx -180 ry 0 rz 180 deg; joints [-138.921, 67.08, -77.449, 138.453, 82.203, 6.856]
  Call Extruder(397.70039)
  MoveL 6944 to (-28.43, 164.09, 97.46) mm, rotated rx -180 ry 0 rz 180 deg; joints [-138.95, 67.086, -77.442, 138.483, 82.208, 6.844]
  Set speed (130.0 mm/s)
  MoveL 6945 to (-31.76, 163.31, 97.46) mm, rotated rx -180 ry 0 rz 180 deg; joints [-139.581, 67.208, -77.308, 139.139, 82.328, 6.588]
  MoveL 6946 to (-31.76, 163.31, 106.87) mm, rotated rx 180 ry 0 rz -180 deg; joints [-139.581, 68.569, -79.157, 139.095, 81.958, 6.911]
  Call Extruder(395.70039)
  Set speed (40.0 mm/s)
  MoveL 6947 to (-31.76, 163.31, 106.87) mm, rotated rx 180 ry 0 rz -180 deg; joints [-139.581, 68.569, -79.157, 139.095, 81.958, 6.911]
  Call Extruder(0.00000)
  Set speed (130.0 mm/s)
  MoveL 6948 to (-31.64, 163.21, 106.87) mm, rotated rx -180 ry 0 rz -180 deg; joints [-139.581, 68.559, -79.168, 139.092, 81.943, 6.924]
  Call Extruder(2.00000)
  Set speed (40.0 mm/s)
  MoveL 6949 to (-31.64, 163.21, 106.87) mm, rotated rx -180 ry 0 rz -180 deg; joints [-139.581, 68.559, -79.168, 139.092, 81.943, 6.924]
  Set speed (30.0 mm/s)
  MoveL 6950 to (-31.64, 163.21, 106.87) mm, rotated rx -180 ry 0 rz -180 deg; joints [-139.581, 68.559, -79.168, 139.092, 81.943, 6.924]
  Call Extruder(2.18198)
  MoveL 6951 to (-31.93, 163.09, 106.87) mm, rotated rx -180 ry 0 rz -180 deg; joints [-139.645, 68.568, -79.158, 139.158, 81.949, 6.903]
  MoveL 6952 to (-31.93, 163.09, 106.87) mm, rotated rx -180 ry 0 rz -180 deg; joints [-139.645, 68.568, -79.158, 139.158, 81.949, 6.903]
  Call Extruder(2.36471)
  MoveL 6953 to (-32.22, 162.96, 106.87) mm, rotated rx -180 ry 0 rz 180 deg; joints [-139.709, 68.577, -79.149, 139.224, 81.955, 6.882]
  MoveL 6954 to (-32.22, 162.96, 106.87) mm, rotated rx -180 ry 0 rz 180 deg; joints [-139.709, 68.577, -79.149, 139.224, 81.955, 6.882]
  Call Extruder(2.53513)
  MoveL 6955 to (-32.49, 162.85, 106.87) mm, rotated rx -180 ry 0 rz 180 deg; joints [-139.768, 68.585, -79.14, 139.285, 81.961, 6.862]
  MoveL 6956 to (-32.49, 162.85, 106.87) mm, rotated rx -180 ry 0 rz 180 deg; joints [-139.768, 68.585, -79.14, 139.285, 81.961, 6.862]
  Call Extruder(2.69310)
  MoveL 6957 to (-32.74, 162.74, 106.87) mm, rotated rx -180 ry 0 rz 180 deg; joints [-139.823, 68.592, -79.132, 139.342, 81.967, 6.844]
  MoveL 6958 to (-32.74, 162.74, 106.87) mm, rotated rx -180 ry 0 rz 180 deg; joints [-139.823, 68.592, -79.132, 139.342, 81.967, 6.844]
  Call Extruder(2.85168)
  MoveL 6959 to (-32.99, 162.64, 106.87) mm, rotated rx -180 ry 0 rz 180 deg; joints [-139.878, 68.6, -79.123, 139.399, 81.972, 6.826]
  MoveL 6960 to (-32.99, 162.64, 106.87) mm, rotated rx -180 ry 0 rz 180 deg; joints [-139.878, 68.6, -79.123, 139.399, 81.972, 6.826]
  Call Extruder(3.05785)
  MoveL 6961 to (-33.29, 162.46, 106.87) mm, rotated rx -180 ry 0 rz 180 deg; joints [-139.953, 68.607, -79.115, 139.475, 81.975, 6.806]
  MoveL 6962 to (-33.29, 162.46, 106.87) mm, rotated rx -180 ry 0 rz 180 deg; joints [-139.953, 68.607, -79.115, 139.475, 81.975, 6.806]
  Call Extruder(3.26479)
  MoveL 6963 to (-33.6, 162.29, 106.87) mm, rotated rx 180 ry 0 rz 180 deg; joints [-140.028, 68.615, -79.107, 139.552, 81.978, 6.785]
  MoveL 6964 to (-33.6, 162.29, 106.87) mm, rotated rx 180 ry 0 rz 180 deg; joints [-140.028, 68.615, -79.107, 139.552, 81.978, 6.785]
  Call Extruder(3.47251)
  MoveL 6965 to (-33.9, 162.11, 106.87) mm, rotated rx 180 ry 0 rz -180 deg; joints [-140.103, 68.622, -79.099, 139.628, 81.981, 6.764]
  MoveL 6966 to (-33.9, 162.11, 106.87) mm, rotated rx 180 ry 0 rz -180 deg; joints [-140.103, 68.622, -79.099, 139.628, 81.981, 6.764]
  Call Extruder(3.68101)
  MoveL 6967 to (-34.21, 161.94, 106.87) mm, rotated rx -180 ry 0 rz -180 deg; joints [-140.178, 68.629, -79.091, 139.705, 81.984, 6.744]
  MoveL 6968 to (-34.21, 161.94, 106.87) mm, rotated rx -180 ry 0 rz -180 deg; joints [-140.178, 68.629, -79.091, 139.705, 81.984, 6.744]
  Call Extruder(3.86055)
  MoveL 6969 to (-34.45, 161.76, 106.87) mm, rotated rx 180 ry 0 rz 180 deg; joints [-140.244, 68.634, -79.086, 139.772, 81.983, 6.728]
  MoveL 6970 to (-34.45, 161.76, 106.87) mm, rotated rx 180 ry 0 rz 180 deg; joints [-140.244, 68.634, -79.086, 139.772, 81.983, 6.728]
  Call Extruder(4.19399)
  MoveL 6971 to (-34.9, 161.43, 106.87) mm, rotated rx -180 ry 0 rz -180 deg; joints [-140.366, 68.643, -79.077, 139.896, 81.982, 6.7]
  MoveL 6972 to (-34.9, 161.43, 106.87) mm, rotated rx -180 ry 0 rz -180 deg; joints [-140.366, 68.643, -79.077, 139.896, 81.982, 6.7]
  Call Extruder(4.52861)
  MoveL 6973 to (-35.35, 161.1, 106.87) mm, rotated rx 180 ry 0 rz 180 deg; joints [-140.489, 68.651, -79.067, 140.02, 81.982, 6.671]
  Call Extruder(5.35652)
  MoveL 6974 to (-36.39, 160.19, 106.87) mm, rotated rx -180 ry 0 rz -180 deg; joints [-140.797, 68.665, -79.052, 140.332, 81.968, 6.609]
  Call Extruder(6.18445)
  MoveL 6975 to (-37.3, 159.15, 106.87) mm, rotated rx -180 ry 0 rz 180 deg; joints [-141.109, 68.668, -79.048, 140.646, 81.938, 6.561]
  Call Extruder(6.35176)
  MoveL 6976 to (-37.47, 158.93, 106.87) mm, rotated rx -180 ry 0 rz 180 deg; joints [-141.172, 68.667, -79.049, 140.709, 81.929, 6.553]
  MoveL 6977 to (-37.47, 158.93, 106.87) mm, rotated rx -180 ry 0 rz 180 deg; joints [-141.172, 68.667, -79.049, 140.709, 81.929, 6.553]
  Call Extruder(6.68519)
  MoveL 6978 to (-37.8, 158.48, 106.87) mm, rotated rx -180 ry 0 rz -180 deg; joints [-141.298, 68.666, -79.051, 140.835, 81.912, 6.537]
  MoveL 6979 to (-37.8, 158.48, 106.87) mm, rotated rx -180 ry 0 rz -180 deg; joints [-141.298, 68.666, -79.051, 140.835, 81.912, 6.537]
  Call Extruder(7.01743)
  MoveL 6980 to (-38.12, 158.03, 106.87) mm, rotated rx -180 ry 0 rz 180 deg; joints [-141.424, 68.664, -79.053, 140.961, 81.896, 6.522]
  MoveL 6981 to (-38.12, 158.03, 106.87) mm, rotated rx -180 ry 0 rz 180 deg; joints [-141.424, 68.664, -79.053, 140.961, 81.896, 6.522]
  Call Extruder(7.13511)
  MoveL 6982 to (-38.22, 157.85, 106.87) mm, rotated rx -180 ry 0 rz 180 deg; joints [-141.468, 68.662, -79.055, 141.005, 81.888, 6.518]
  MoveL 6983 to (-38.22, 157.85, 106.87) mm, rotated rx -180 ry 0 rz 180 deg; joints [-141.468, 68.662, -79.055, 141.005, 81.888, 6.518]
  Call Extruder(7.34283)
  MoveL 6984 to (-38.4, 157.55, 106.87) mm, rotated rx -180 ry 0 rz -180 deg; joints [-141.547, 68.659, -79.058, 141.084, 81.874, 6.511]
  MoveL 6985 to (-38.4, 157.55, 106.87) mm, rotated rx -180 ry 0 rz -180 deg; joints [-141.547, 68.659, -79.058, 141.084, 81.874, 6.511]
  Call Extruder(7.54978)
  MoveL 6986 to (-38.57, 157.25, 106.87) mm, rotated rx 180 ry 0 rz 180 deg; joints [-141.625, 68.656, -79.062, 141.162, 81.86, 6.504]
  MoveL 6987 to (-38.57, 157.25, 106.87) mm, rotated rx 180 ry 0 rz 180 deg; joints [-141.625, 68.656, -79.062, 141.162, 81.86, 6.504]
  Call Extruder(7.75595)
  MoveL 6988 to (-38.75, 156.94, 106.87) mm, rotated rx 180 ry 0 rz 180 deg; joints [-141.704, 68.653, -79.065, 141.24, 81.845, 6.497]
  MoveL 6989 to (-38.75, 156.94, 106.87) mm, rotated rx 180 ry 0 rz 180 deg; joints [-141.704, 68.653, -79.065, 141.24, 81.845, 6.497]
  Call Extruder(7.93763)
  MoveL 6990 to (-38.89, 156.67, 106.87) mm, rotated rx -180 ry 0 rz 180 deg; joints [-141.773, 68.649, -79.069, 141.309, 81.832, 6.492]
  MoveL 6991 to (-38.89, 156.67, 106.87) mm, rotated rx -180 ry 0 rz 180 deg; joints [-141.773, 68.649, -79.069, 141.309, 81.832, 6.492]
  Call Extruder(8.09561)
  MoveL 6992 to (-39, 156.42, 106.87) mm, rotated rx 180 ry 0 rz 180 deg; joints [-141.832, 68.645, -79.074, 141.367, 81.818, 6.489]
  MoveL 6993 to (-39, 156.42, 106.87) mm, rotated rx 180 ry 0 rz 180 deg; joints [-141.832, 68.645, -79.074, 141.367, 81.818, 6.489]
  Call Extruder(8.25300)
  MoveL 6994 to (-39.1, 156.17, 106.87) mm, rotated rx -180 ry 0 rz -180 deg; joints [-141.891, 68.641, -79.079, 141.426, 81.804, 6.486]
  MoveL 6995 to (-39.1, 156.17, 106.87) mm, rotated rx -180 ry 0 rz -180 deg; joints [-141.891, 68.641, -79.079, 141.426, 81.804, 6.486]
  Call Extruder(8.43571)
  MoveL 6996 to (-39.23, 155.88, 106.87) mm, rotated rx 180 ry 0 rz -180 deg; joints [-141.96, 68.635, -79.085, 141.494, 81.788, 6.483]
  MoveL 6997 to (-39.23, 155.88, 106.87) mm, rotated rx 180 ry 0 rz -180 deg; joints [-141.96, 68.635, -79.085, 141.494, 81.788, 6.483]
  Call Extruder(8.61768)
  MoveL 6998 to (-39.35, 155.58, 106.87) mm, rotated rx -180 ry 0 rz 180 deg; joints [-142.029, 68.63, -79.09, 141.563, 81.772, 6.48]
  MoveL 6999 to (-39.35, 155.58, 106.87) mm, rotated rx -180 ry 0 rz 180 deg; joints [-142.029, 68.63, -79.09, 141.563, 81.772, 6.48]
  Call Extruder(8.76501)
  MoveL 7000 to (-39.44, 155.34, 106.87) mm, rotated rx 180 ry 0 rz 180 deg; joints [-142.085, 68.626, -79.095, 141.617, 81.758, 6.478]
  MoveL 7001 to (-39.44, 155.34, 106.87) mm, rotated rx 180 ry 0 rz 180 deg; joints [-142.085, 68.626, -79.095, 141.617, 81.758, 6.478]
  Call Extruder(8.87825)
  MoveL 7002 to (-39.5, 155.15, 106.87) mm, rotated rx -180 ry 0 rz -180 deg; joints [-142.127, 68.621, -79.1, 141.659, 81.746, 6.478]
  MoveL 7003 to (-39.5, 155.15, 106.87) mm, rotated rx -180 ry 0 rz -180 deg; joints [-142.127, 68.621, -79.1, 141.659, 81.746, 6.478]
  Call Extruder(8.99104)
  MoveL 7004 to (-39.56, 154.97, 106.87) mm, rotated rx -180 ry 0 rz -180 deg; joints [-142.169, 68.617, -79.104, 141.701, 81.735, 6.477]
  MoveL 7005 to (-39.56, 154.97, 106.87) mm, rotated rx -180 ry 0 rz -180 deg; joints [-142.169, 68.617, -79.104, 141.701, 81.735, 6.477]
  Call Extruder(9.10338)
  MoveL 7006 to (-39.62, 154.78, 106.87) mm, rotated rx -180 ry 0 rz 180 deg; joints [-142.212, 68.613, -79.109, 141.743, 81.723, 6.476]
  MoveL 7007 to (-39.62, 154.78, 106.87) mm, rotated rx -180 ry 0 rz 180 deg; joints [-142.212, 68.613, -79.109, 141.743, 81.723, 6.476]
  Call Extruder(9.21528)
  MoveL 7008 to (-39.68, 154.59, 106.87) mm, rotated rx -180 ry 0 rz -180 deg; joints [-142.254, 68.609, -79.113, 141.784, 81.711, 6.476]
  MoveL 7009 to (-39.68, 154.59, 106.87) mm, rotated rx -180 ry 0 rz -180 deg; joints [-142.254, 68.609, -79.113, 141.784, 81.711, 6.476]
  Call Extruder(9.33668)
  MoveL 7010 to (-39.75, 154.38, 106.87) mm, rotated rx 180 ry 0 rz 180 deg; joints [-142.3, 68.604, -79.118, 141.829, 81.699, 6.475]
  MoveL 7011 to (-39.75, 154.38, 106.87) mm, rotated rx 180 ry 0 rz 180 deg; joints [-142.3, 68.604, -79.118, 141.829, 81.699, 6.475]
  Call Extruder(9.46748)
  MoveL 7012 to (-39.81, 154.16, 106.87) mm, rotated rx 180 ry 0 rz 180 deg; joints [-142.35, 68.599, -79.124, 141.878, 81.685, 6.475]
  MoveL 7013 to (-39.81, 154.16, 106.87) mm, rotated rx 180 ry 0 rz 180 deg; joints [-142.35, 68.599, -79.124, 141.878, 81.685, 6.475]
  Call Extruder(9.59770)
  MoveL 7014 to (-39.88, 153.94, 106.87) mm, rotated rx 180 ry 0 rz 180 deg; joints [-142.399, 68.594, -79.13, 141.927, 81.671, 6.474]
  MoveL 7015 to (-39.88, 153.94, 106.87) mm, rotated rx 180 ry 0 rz 180 deg; joints [-142.399, 68.594, -79.13, 141.927, 81.671, 6.474]
  Call Extruder(9.72737)
  MoveL 7016 to (-39.95, 153.71, 106.87) mm, rotated rx 180 ry 0 rz 180 deg; joints [-142.449, 68.589, -79.135, 141.976, 81.657, 6.473]
  MoveL 7017 to (-39.95, 153.71, 106.87) mm, rotated rx 180 ry 0 rz 180 deg; joints [-142.449, 68.589, -79.135, 141.976, 81.657, 6.473]
  Call Extruder(9.85647)
  MoveL 7018 to (-40.02, 153.49, 106.87) mm, rotated rx 180 ry 0 rz -180 deg; joints [-142.498, 68.584, -79.141, 142.025, 81.643, 6.473]
  MoveL 7019 to (-40.02, 153.49, 106.87) mm, rotated rx 180 ry 0 rz -180 deg; joints [-142.498, 68.584, -79.141, 142.025, 81.643, 6.473]
  Call Extruder(9.97156)
  MoveL 7020 to (-40.06, 153.28, 106.87) mm, rotated rx 180 ry 0 rz 180 deg; joints [-142.541, 68.579, -79.147, 142.067, 81.629, 6.474]
  MoveL 7021 to (-40.06, 153.28, 106.87) mm, rotated rx 180 ry 0 rz 180 deg; joints [-142.541, 68.579, -79.147, 142.067, 81.629, 6.474]
  Call Extruder(10.08619)
  MoveL 7022 to (-40.11, 153.08, 106.87) mm, rotated rx 180 ry 0 rz 180 deg; joints [-142.584, 68.573, -79.153, 142.109, 81.615, 6.474]
  MoveL 7023 to (-40.11, 153.08, 106.87) mm, rotated rx 180 ry 0 rz 180 deg; joints [-142.584, 68.573, -79.153, 142.109, 81.615, 6.474]
  Call Extruder(10.20037)
  MoveL 7024 to (-40.15, 152.88, 106.87) mm, rotated rx 180 ry 0 rz 180 deg; joints [-142.627, 68.568, -79.159, 142.151, 81.601, 6.475]
  MoveL 7025 to (-40.15, 152.88, 106.87) mm, rotated rx 180 ry 0 rz 180 deg; joints [-142.627, 68.568, -79.159, 142.151, 81.601, 6.475]
  Call Extruder(10.31410)
  MoveL 7026 to (-40.2, 152.67, 106.87) mm, rotated rx 180 ry 0 rz -180 deg; joints [-142.671, 68.562, -79.164, 142.194, 81.587, 6.476]
  MoveL 7027 to (-40.2, 152.67, 106.87) mm, rotated rx 180 ry 0 rz -180 deg; joints [-142.671, 68.562, -79.164, 142.194, 81.587, 6.476]
  Call Extruder(10.43953)
  MoveL 7028 to (-40.24, 152.44, 106.87) mm, rotated rx -180 ry 0 rz -180 deg; joints [-142.718, 68.556, -79.171, 142.24, 81.572, 6.477]
  MoveL 7029 to (-40.24, 152.44, 106.87) mm, rotated rx -180 ry 0 rz -180 deg; joints [-142.718, 68.556, -79.171, 142.24, 81.572, 6.477]
  Call Extruder(10.57651)
  MoveL 7030 to (-40.29, 152.2, 106.87) mm, rotated rx -180 ry 0 rz -180 deg; joints [-142.77, 68.549, -79.179, 142.291, 81.555, 6.478]
  MoveL 7031 to (-40.29, 152.2, 106.87) mm, rotated rx -180 ry 0 rz -180 deg; joints [-142.77, 68.549, -79.179, 142.291, 81.555, 6.478]
  Call Extruder(10.71287)
  MoveL 7032 to (-40.34, 151.95, 106.87) mm, rotated rx -180 ry 0 rz -180 deg; joints [-142.822, 68.542, -79.186, 142.342, 81.537, 6.479]
  MoveL 7033 to (-40.34, 151.95, 106.87) mm, rotated rx -180 ry 0 rz -180 deg; joints [-142.822, 68.542, -79.186, 142.342, 81.537, 6.479]
  Call Extruder(10.84863)
  MoveL 7034 to (-40.39, 151.7, 106.87) mm, rotated rx 180 ry 0 rz 180 deg; joints [-142.874, 68.535, -79.193, 142.393, 81.52, 6.48]
  MoveL 7035 to (-40.39, 151.7, 106.87) mm, rotated rx 180 ry 0 rz 180 deg; joints [-142.874, 68.535, -79.193, 142.393, 81.52, 6.48]
  Call Extruder(10.98377)
  MoveL 7036 to (-40.44, 151.45, 106.87) mm, rotated rx -180 ry 0 rz 180 deg; joints [-142.926, 68.529, -79.201, 142.444, 81.503, 6.481]
  MoveL 7037 to (-40.44, 151.45, 106.87) mm, rotated rx -180 ry 0 rz 180 deg; joints [-142.926, 68.529, -79.201, 142.444, 81.503, 6.481]
  Call Extruder(11.11831)
  MoveL 7038 to (-40.49, 151.2, 106.87) mm, rotated rx -180 ry 0 rz 180 deg; joints [-142.978, 68.522, -79.208, 142.495, 81.486, 6.482]
  MoveL 7039 to (-40.49, 151.2, 106.87) mm, rotated rx -180 ry 0 rz 180 deg; joints [-142.978, 68.522, -79.208, 142.495, 81.486, 6.482]
  Call Extruder(11.25223)
  MoveL 7040 to (-40.54, 150.95, 106.87) mm, rotated rx 180 ry 0 rz 180 deg; joints [-143.031, 68.515, -79.216, 142.546, 81.469, 6.483]
  MoveL 7041 to (-40.54, 150.95, 106.87) mm, rotated rx 180 ry 0 rz 180 deg; joints [-143.031, 68.515, -79.216, 142.546, 81.469, 6.483]
  Call Extruder(11.40009)
  MoveL 7042 to (-40.59, 150.67, 106.87) mm, rotated rx 180 ry 0 rz -180 deg; joints [-143.088, 68.507, -79.224, 142.603, 81.449, 6.485]
  MoveL 7043 to (-40.59, 150.67, 106.87) mm, rotated rx 180 ry 0 rz -180 deg; joints [-143.088, 68.507, -79.224, 142.603, 81.449, 6.485]
  Call Extruder(11.56181)
  MoveL 7044 to (-40.64, 150.37, 106.87) mm, rotated rx -180 ry 0 rz 180 deg; joints [-143.15, 68.498, -79.234, 142.664, 81.427, 6.487]
  MoveL 7045 to (-40.64, 150.37, 106.87) mm, rotated rx -180 ry 0 rz 180 deg; joints [-143.15, 68.498, -79.234, 142.664, 81.427, 6.487]
  Call Extruder(11.72281)
  MoveL 7046 to (-40.69, 150.06, 106.87) mm, rotated rx 180 ry 0 rz 180 deg; joints [-143.213, 68.489, -79.243, 142.725, 81.406, 6.489]
  MoveL 7047 to (-40.69, 150.06, 106.87) mm, rotated rx 180 ry 0 rz 180 deg; joints [-143.213, 68.489, -79.243, 142.725, 81.406, 6.489]
  Call Extruder(11.88308)
  MoveL 7048 to (-40.74, 149.76, 106.87) mm, rotated rx 180 ry 0 rz 180 deg; joints [-143.276, 68.48, -79.253, 142.786, 81.384, 6.491]
  MoveL 7049 to (-40.74, 149.76, 106.87) mm, rotated rx 180 ry 0 rz 180 deg; joints [-143.276, 68.48, -79.253, 142.786, 81.384, 6.491]
  Call Extruder(12.04262)
  MoveL 7050 to (-40.78, 149.45, 106.87) mm, rotated rx 180 ry 0 rz 180 deg; joints [-143.338, 68.471, -79.262, 142.847, 81.362, 6.493]
  MoveL 7051 to (-40.78, 149.45, 106.87) mm, rotated rx 180 ry 0 rz 180 deg; joints [-143.338, 68.471, -79.262, 142.847, 81.362, 6.493]
  Call Extruder(12.20143)
  MoveL 7052 to (-40.83, 149.14, 106.87) mm, rotated rx -180 ry 0 rz 180 deg; joints [-143.401, 68.462, -79.272, 142.909, 81.34, 6.494]
  MoveL 7053 to (-40.83, 149.14, 106.87) mm, rotated rx -180 ry 0 rz 180 deg; joints [-143.401, 68.462, -79.272, 142.909, 81.34, 6.494]
  Call Extruder(12.38010)
  MoveL 7054 to (-40.88, 148.8, 106.87) mm, rotated rx -180 ry 0 rz -180 deg; joints [-143.471, 68.452, -79.283, 142.977, 81.315, 6.497]
  MoveL 7055 to (-40.88, 148.8, 106.87) mm, rotated rx -180 ry 0 rz -180 deg; joints [-143.471, 68.452, -79.283, 142.977, 81.315, 6.497]
  Call Extruder(12.57854)
  MoveL 7056 to (-40.92, 148.41, 106.87) mm, rotated rx -180 ry 0 rz 180 deg; joints [-143.549, 68.44, -79.296, 143.053, 81.286, 6.5]
  MoveL 7057 to (-40.92, 148.41, 106.87) mm, rotated rx -180 ry 0 rz 180 deg; joints [-143.549, 68.44, -79.296, 143.053, 81.286, 6.5]
  Call Extruder(12.77611)
  MoveL 7058 to (-40.97, 148.02, 106.87) mm, rotated rx -180 ry 0 rz -180 deg; joints [-143.627, 68.428, -79.309, 143.129, 81.258, 6.503]
  MoveL 7059 to (-40.97, 148.02, 106.87) mm, rotated rx -180 ry 0 rz -180 deg; joints [-143.627, 68.428, -79.309, 143.129, 81.258, 6.503]
  Call Extruder(12.97282)
  MoveL 7060 to (-41.02, 147.63, 106.87) mm, rotated rx 180 ry 0 rz 180 deg; joints [-143.705, 68.416, -79.321, 143.205, 81.229, 6.507]
  MoveL 7061 to (-41.02, 147.63, 106.87) mm, rotated rx 180 ry 0 rz 180 deg; joints [-143.705, 68.416, -79.321, 143.205, 81.229, 6.507]
  Call Extruder(13.16865)
  MoveL 7062 to (-41.06, 147.25, 106.87) mm, rotated rx 180 ry 0 rz 180 deg; joints [-143.783, 68.404, -79.334, 143.281, 81.2, 6.51]
  MoveL 7063 to (-41.06, 147.25, 106.87) mm, rotated rx 180 ry 0 rz 180 deg; joints [-143.783, 68.404, -79.334, 143.281, 81.2, 6.51]
  Call Extruder(13.46405)
  MoveL 7064 to (-41.11, 146.66, 106.87) mm, rotated rx -180 ry 0 rz -180 deg; joints [-143.899, 68.384, -79.355, 143.394, 81.155, 6.516]
  MoveL 7065 to (-41.11, 146.66, 106.87) mm, rotated rx -180 ry 0 rz -180 deg; joints [-143.899, 68.384, -79.355, 143.394, 81.155, 6.516]
  Call Extruder(13.75812)
  MoveL 7066 to (-41.15, 146.07, 106.87) mm, rotated rx -180 ry 0 rz 180 deg; joints [-144.015, 68.365, -79.375, 143.507, 81.11, 6.522]
  MoveL 7067 to (-41.15, 146.07, 106.87) mm, rotated rx -180 ry 0 rz 180 deg; joints [-144.015, 68.365, -79.375, 143.507, 81.11, 6.522]
  Call Extruder(14.05086)
  MoveL 7068 to (-41.2, 145.48, 106.87) mm, rotated rx 180 ry 0 rz 180 deg; joints [-144.131, 68.345, -79.395, 143.621, 81.065, 6.527]
  MoveL 7069 to (-41.2, 145.48, 106.87) mm, rotated rx 180 ry 0 rz 180 deg; joints [-144.131, 68.345, -79.395, 143.621, 81.065, 6.527]
  Call Extruder(14.62431)
  MoveL 7070 to (-41.25, 144.32, 106.87) mm, rotated rx -180 ry 0 rz -180 deg; joints [-144.355, 68.305, -79.437, 143.838, 80.973, 6.542]
  MoveL 7071 to (-41.25, 144.32, 106.87) mm, rotated rx -180 ry 0 rz -180 deg; joints [-144.355, 68.305, -79.437, 143.838, 80.973, 6.542]
  Call Extruder(15.33827)
  MoveL 7072 to (-41.29, 142.86, 106.87) mm, rotated rx 180 ry 0 rz 180 deg; joints [-144.635, 68.254, -79.49, 144.11, 80.857, 6.559]
  Call Extruder(57.40309)
  MoveL 7073 to (-41.29, 57.14, 106.87) mm, rotated rx -180 ry 0 rz -180 deg; joints [-164.153, 65.648, -81.67, 163.546, 74.602, 4.484]
  Call Extruder(57.83165)
  MoveL 7074 to (-41.27, 56.26, 106.87) mm, rotated rx -180 ry 0 rz -180 deg; joints [-164.382, 65.629, -81.683, 163.781, 74.554, 4.43]
  MoveL 7075 to (-41.27, 56.26, 106.87) mm, rotated rx -180 ry 0 rz -180 deg; joints [-164.382, 65.629, -81.683, 163.781, 74.554, 4.43]
  Call Extruder(58.11773)
  MoveL 7076 to (-41.25, 55.68, 106.87) mm, rotated rx -180 ry 0 rz 180 deg; joints [-164.534, 65.616, -81.692, 163.936, 74.521, 4.395]
  MoveL 7077 to (-41.25, 55.68, 106.87) mm, rotated rx -180 ry 0 rz 180 deg; joints [-164.534, 65.616, -81.692, 163.936, 74.521, 4.395]
  Call Extruder(58.69247)
  MoveL 7078 to (-41.2, 54.52, 106.87) mm, rotated rx -180 ry 0 rz 180 deg; joints [-164.838, 65.589, -81.71, 164.248, 74.455, 4.323]
  MoveL 7079 to (-41.2, 54.52, 106.87) mm, rotated rx -180 ry 0 rz 180 deg; joints [-164.838, 65.589, -81.71, 164.248, 74.455, 4.323]
  Call Extruder(58.98587)
  MoveL 7080 to (-41.15, 53.93, 106.87) mm, rotated rx 180 ry 0 rz 180 deg; joints [-164.992, 65.574, -81.72, 164.405, 74.419, 4.287]
  MoveL 7081 to (-41.15, 53.93, 106.87) mm, rotated rx 180 ry 0 rz 180 deg; joints [-164.992, 65.574, -81.72, 164.405, 74.419, 4.287]
  Call Extruder(59.28060)
  MoveL 7082 to (-41.11, 53.34, 106.87) mm, rotated rx -180 ry 0 rz 180 deg; joints [-165.145, 65.559, -81.73, 164.562, 74.384, 4.252]
  MoveL 7083 to (-41.11, 53.34, 106.87) mm, rotated rx -180 ry 0 rz 180 deg; joints [-165.145, 65.559, -81.73, 164.562, 74.384, 4.252]
  Call Extruder(59.57666)
  MoveL 7084 to (-41.06, 52.75, 106.87) mm, rotated rx 180 ry 0 rz 180 deg; joints [-165.299, 65.545, -81.74, 164.719, 74.349, 4.215]
  MoveL 7085 to (-41.06, 52.75, 106.87) mm, rotated rx 180 ry 0 rz 180 deg; joints [-165.299, 65.545, -81.74, 164.719, 74.349, 4.215]
  Call Extruder(59.77293)
  MoveL 7086 to (-41.02, 52.36, 106.87) mm, rotated rx -180 ry 0 rz -180 deg; joints [-165.399, 65.534, -81.747, 164.822, 74.324, 4.192]
  MoveL 7087 to (-41.02, 52.36, 106.87) mm, rotated rx -180 ry 0 rz -180 deg; joints [-165.399, 65.534, -81.747, 164.822, 74.324, 4.192]
  Call Extruder(59.97007)
  MoveL 7088 to (-40.97, 51.98, 106.87) mm, rotated rx -180 ry 0 rz -180 deg; joints [-165.499, 65.523, -81.754, 164.924, 74.3, 4.169]
  MoveL 7089 to (-40.97, 51.98, 106.87) mm, rotated rx -180 ry 0 rz -180 deg; joints [-165.499, 65.523, -81.754, 164.924, 74.3, 4.169]
  Call Extruder(60.16808)
  MoveL 7090 to (-40.92, 51.59, 106.87) mm, rotated rx -180 ry 0 rz 180 deg; joints [-165.6, 65.513, -81.761, 165.027, 74.275, 4.146]
  MoveL 7091 to (-40.92, 51.59, 106.87) mm, rotated rx -180 ry 0 rz 180 deg; joints [-165.6, 65.513, -81.761, 165.027, 74.275, 4.146]
  Call Extruder(60.36695)
  MoveL 7092 to (-40.88, 51.2, 106.87) mm, rotated rx -180 ry 0 rz 180 deg; joints [-165.7, 65.502, -81.768, 165.13, 74.251, 4.122]
  MoveL 7093 to (-40.88, 51.2, 106.87) mm, rotated rx -180 ry 0 rz 180 deg; joints [-165.7, 65.502, -81.768, 165.13, 74.251, 4.122]
  Call Extruder(60.54603)
  MoveL 7094 to (-40.83, 50.86, 106.87) mm, rotated rx -180 ry 0 rz -180 deg; joints [-165.79, 65.492, -81.775, 165.222, 74.229, 4.101]
  MoveL 7095 to (-40.83, 50.86, 106.87) mm, rotated rx -180 ry 0 rz -180 deg; joints [-165.79, 65.492, -81.775, 165.222, 74.229, 4.101]
  Call Extruder(60.70521)
  MoveL 7096 to (-40.78, 50.55, 106.87) mm, rotated rx 180 ry 0 rz -180 deg; joints [-165.869, 65.483, -81.781, 165.302, 74.208, 4.083]
  MoveL 7097 to (-40.78, 50.55, 106.87) mm, rotated rx 180 ry 0 rz -180 deg; joints [-165.869, 65.483, -81.781, 165.302, 74.208, 4.083]
  Call Extruder(60.86512)
  MoveL 7098 to (-40.74, 50.24, 106.87) mm, rotated rx -180 ry 0 rz 180 deg; joints [-165.948, 65.473, -81.787, 165.383, 74.188, 4.065]
  MoveL 7099 to (-40.74, 50.24, 106.87) mm, rotated rx -180 ry 0 rz 180 deg; joints [-165.948, 65.473, -81.787, 165.383, 74.188, 4.065]
  Call Extruder(61.02575)
  MoveL 7100 to (-40.69, 49.94, 106.87) mm, rotated rx 180 ry 0 rz 180 deg; joints [-166.026, 65.464, -81.793, 165.463, 74.167, 4.047]
  MoveL 7101 to (-40.69, 49.94, 106.87) mm, rotated rx 180 ry 0 rz 180 deg; joints [-166.026, 65.464, -81.793, 165.463, 74.167, 4.047]
  Call Extruder(61.18711)
  MoveL 7102 to (-40.64, 49.63, 106.87) mm, rotated rx 180 ry 0 rz -180 deg; joints [-166.105, 65.455, -81.799, 165.544, 74.147, 4.028]
  MoveL 7103 to (-40.64, 49.63, 106.87) mm, rotated rx 180 ry 0 rz -180 deg; joints [-166.105, 65.455, -81.799, 165.544, 74.147, 4.028]
  Call Extruder(61.34920)
  MoveL 7104 to (-40.59, 49.33, 106.87) mm, rotated rx 180 ry 0 rz 180 deg; joints [-166.184, 65.446, -81.805, 165.625, 74.127, 4.01]
  MoveL 7105 to (-40.59, 49.33, 106.87) mm, rotated rx 180 ry 0 rz 180 deg; joints [-166.184, 65.446, -81.805, 165.625, 74.127, 4.01]
  Call Extruder(61.49740)
  MoveL 7106 to (-40.54, 49.05, 106.87) mm, rotated rx 180 ry 0 rz 180 deg; joints [-166.256, 65.437, -81.811, 165.698, 74.108, 3.993]
  MoveL 7107 to (-40.54, 49.05, 106.87) mm, rotated rx 180 ry 0 rz 180 deg; joints [-166.256, 65.437, -81.811, 165.698, 74.108, 3.993]
  Call Extruder(61.63163)
  MoveL 7108 to (-40.49, 48.8, 106.87) mm, rotated rx 180 ry 0 rz 180 deg; joints [-166.32, 65.429, -81.816, 165.764, 74.09, 3.978]
  MoveL 7109 to (-40.49, 48.8, 106.87) mm, rotated rx 180 ry 0 rz 180 deg; joints [-166.32, 65.429, -81.816, 165.764, 74.09, 3.978]
  Call Extruder(61.76647)
  MoveL 7110 to (-40.44, 48.55, 106.87) mm, rotated rx -180 ry 0 rz -180 deg; joints [-166.384, 65.421, -81.821, 165.829, 74.073, 3.964]
  MoveL 7111 to (-40.44, 48.55, 106.87) mm, rotated rx -180 ry 0 rz -180 deg; joints [-166.384, 65.421, -81.821, 165.829, 74.073, 3.964]
  Call Extruder(61.90192)
  MoveL 7112 to (-40.39, 48.3, 106.87) mm, rotated rx -180 ry 0 rz -180 deg; joints [-166.448, 65.413, -81.827, 165.895, 74.056, 3.949]
  MoveL 7113 to (-40.39, 48.3, 106.87) mm, rotated rx -180 ry 0 rz -180 deg; joints [-166.448, 65.413, -81.827, 165.895, 74.056, 3.949]
  Call Extruder(62.03798)
  MoveL 7114 to (-40.34, 48.05, 106.87) mm, rotated rx 180 ry 0 rz 180 deg; joints [-166.512, 65.405, -81.832, 165.96, 74.038, 3.934]
  MoveL 7115 to (-40.34, 48.05, 106.87) mm, rotated rx 180 ry 0 rz 180 deg; joints [-166.512, 65.405, -81.832, 165.96, 74.038, 3.934]
  Call Extruder(62.17465)
  MoveL 7116 to (-40.29, 47.8, 106.87) mm, rotated rx 180 ry 0 rz 180 deg; joints [-166.576, 65.397, -81.837, 166.026, 74.021, 3.919]
  MoveL 7117 to (-40.29, 47.8, 106.87) mm, rotated rx 180 ry 0 rz 180 deg; joints [-166.576, 65.397, -81.837, 166.026, 74.021, 3.919]
  Call Extruder(62.31193)
  MoveL 7118 to (-40.24, 47.56, 106.87) mm, rotated rx -180 ry 0 rz 180 deg; joints [-166.641, 65.389, -81.843, 166.092, 74.003, 3.904]
  MoveL 7119 to (-40.24, 47.56, 106.87) mm, rotated rx -180 ry 0 rz 180 deg; joints [-166.641, 65.389, -81.843, 166.092, 74.003, 3.904]
  Call Extruder(62.43760)
  MoveL 7120 to (-40.2, 47.33, 106.87) mm, rotated rx -180 ry 0 rz -180 deg; joints [-166.699, 65.381, -81.847, 166.151, 73.987, 3.89]
  MoveL 7121 to (-40.2, 47.33, 106.87) mm, rotated rx -180 ry 0 rz -180 deg; joints [-166.699, 65.381, -81.847, 166.151, 73.987, 3.89]
  Call Extruder(62.55156)
  MoveL 7122 to (-40.15, 47.12, 106.87) mm, rotated rx -180 ry 0 rz 180 deg; joints [-166.751, 65.374, -81.852, 166.205, 73.973, 3.878]
  MoveL 7123 to (-40.15, 47.12, 106.87) mm, rotated rx -180 ry 0 rz 180 deg; joints [-166.751, 65.374, -81.852, 166.205, 73.973, 3.878]
  Call Extruder(62.66597)
  MoveL 7124 to (-40.11, 46.92, 106.87) mm, rotated rx -180 ry 0 rz 180 deg; joints [-166.804, 65.367, -81.856, 166.259, 73.958, 3.866]
  MoveL 7125 to (-40.11, 46.92, 106.87) mm, rotated rx -180 ry 0 rz 180 deg; joints [-166.804, 65.367, -81.856, 166.259, 73.958, 3.866]
  Call Extruder(62.78083)
  MoveL 7126 to (-40.06, 46.72, 106.87) mm, rotated rx 180 ry 0 rz -180 deg; joints [-166.857, 65.36, -81.861, 166.313, 73.944, 3.853]
  MoveL 7127 to (-40.06, 46.72, 106.87) mm, rotated rx 180 ry 0 rz -180 deg; joints [-166.857, 65.36, -81.861, 166.313, 73.944, 3.853]
  Call Extruder(62.89614)
  MoveL 7128 to (-40.02, 46.51, 106.87) mm, rotated rx -180 ry 0 rz -180 deg; joints [-166.909, 65.354, -81.865, 166.367, 73.929, 3.841]
  MoveL 7129 to (-40.02, 46.51, 106.87) mm, rotated rx -180 ry 0 rz -180 deg; joints [-166.909, 65.354, -81.865, 166.367, 73.929, 3.841]
  Call Extruder(63.02552)
  MoveL 7130 to (-39.95, 46.29, 106.87) mm, rotated rx -180 ry 0 rz -180 deg; joints [-166.966, 65.345, -81.871, 166.424, 73.911, 3.828]
  MoveL 7131 to (-39.95, 46.29, 106.87) mm, rotated rx -180 ry 0 rz -180 deg; joints [-166.966, 65.345, -81.871, 166.424, 73.911, 3.828]
  Call Extruder(63.15547)
  MoveL 7132 to (-39.88, 46.06, 106.87) mm, rotated rx -180 ry 0 rz -180 deg; joints [-167.022, 65.336, -81.877, 166.482, 73.893, 3.816]
  MoveL 7133 to (-39.88, 46.06, 106.87) mm, rotated rx -180 ry 0 rz -180 deg; joints [-167.022, 65.336, -81.877, 166.482, 73.893, 3.816]
  Call Extruder(63.28598)
  MoveL 7134 to (-39.82, 45.84, 106.87) mm, rotated rx -180 ry 0 rz -180 deg; joints [-167.079, 65.327, -81.882, 166.54, 73.875, 3.803]
  MoveL 7135 to (-39.82, 45.84, 106.87) mm, rotated rx -180 ry 0 rz -180 deg; joints [-167.079, 65.327, -81.882, 166.54, 73.875, 3.803]
  Call Extruder(63.41705)
  MoveL 7136 to (-39.75, 45.62, 106.87) mm, rotated rx -180 ry 0 rz 180 deg; joints [-167.136, 65.318, -81.888, 166.598, 73.857, 3.79]
  MoveL 7137 to (-39.75, 45.62, 106.87) mm, rotated rx -180 ry 0 rz 180 deg; joints [-167.136, 65.318, -81.888, 166.598, 73.857, 3.79]
  Call Extruder(63.53870)
  MoveL 7138 to (-39.68, 45.41, 106.87) mm, rotated rx 180 ry 0 rz 180 deg; joints [-167.188, 65.31, -81.894, 166.651, 73.841, 3.778]
  MoveL 7139 to (-39.68, 45.41, 106.87) mm, rotated rx 180 ry 0 rz 180 deg; joints [-167.188, 65.31, -81.894, 166.651, 73.841, 3.778]
  Call Extruder(63.65082)
  MoveL 7140 to (-39.62, 45.22, 106.87) mm, rotated rx -180 ry 0 rz 180 deg; joints [-167.235, 65.302, -81.899, 166.7, 73.825, 3.768]
  MoveL 7141 to (-39.62, 45.22, 106.87) mm, rotated rx -180 ry 0 rz 180 deg; joints [-167.235, 65.302, -81.899, 166.7, 73.825, 3.768]
  Call Extruder(63.76339)
  MoveL 7142 to (-39.56, 45.03, 106.87) mm, rotated rx 180 ry 0 rz 180 deg; joints [-167.283, 65.294, -81.903, 166.749, 73.809, 3.757]
  MoveL 7143 to (-39.56, 45.03, 106.87) mm, rotated rx 180 ry 0 rz 180 deg; joints [-167.283, 65.294, -81.903, 166.749, 73.809, 3.757]
  Call Extruder(63.87640)
  MoveL 7144 to (-39.5, 44.85, 106.87) mm, rotated rx 180 ry 0 rz 180 deg; joints [-167.331, 65.286, -81.908, 166.797, 73.794, 3.746]
  MoveL 7145 to (-39.5, 44.85, 106.87) mm, rotated rx 180 ry 0 rz 180 deg; joints [-167.331, 65.286, -81.908, 166.797, 73.794, 3.746]
  Call Extruder(63.98986)
  MoveL 7146 to (-39.44, 44.66, 106.87) mm, rotated rx 180 ry 0 rz -180 deg; joints [-167.379, 65.279, -81.913, 166.846, 73.778, 3.735]
  MoveL 7147 to (-39.44, 44.66, 106.87) mm, rotated rx 180 ry 0 rz -180 deg; joints [-167.379, 65.279, -81.913, 166.846, 73.778, 3.735]
  Call Extruder(64.13750)
  MoveL 7148 to (-39.35, 44.42, 106.87) mm, rotated rx -180 ry 0 rz 180 deg; joints [-167.439, 65.268, -81.92, 166.908, 73.757, 3.722]
  MoveL 7149 to (-39.35, 44.42, 106.87) mm, rotated rx -180 ry 0 rz 180 deg; joints [-167.439, 65.268, -81.92, 166.908, 73.757, 3.722]
  Call Extruder(64.31984)
  MoveL 7150 to (-39.22, 44.12, 106.87) mm, rotated rx 180 ry 0 rz 180 deg; joints [-167.512, 65.254, -81.929, 166.982, 73.73, 3.706]
  MoveL 7151 to (-39.22, 44.12, 106.87) mm, rotated rx 180 ry 0 rz 180 deg; joints [-167.512, 65.254, -81.929, 166.982, 73.73, 3.706]
  Call Extruder(64.50294)
  MoveL 7152 to (-39.11, 43.83, 106.87) mm, rotated rx -180 ry 0 rz -180 deg; joints [-167.584, 65.24, -81.938, 167.056, 73.703, 3.69]
  MoveL 7153 to (-39.11, 43.83, 106.87) mm, rotated rx -180 ry 0 rz -180 deg; joints [-167.584, 65.24, -81.938, 167.056, 73.703, 3.69]
  Call Extruder(64.66062)
  MoveL 7154 to (-39, 43.58, 106.87) mm, rotated rx 180 ry 0 rz 180 deg; joints [-167.646, 65.228, -81.946, 167.119, 73.68, 3.677]
  MoveL 7155 to (-39, 43.58, 106.87) mm, rotated rx 180 ry 0 rz 180 deg; joints [-167.646, 65.228, -81.946, 167.119, 73.68, 3.677]
  Call Extruder(64.81891)
  MoveL 7156 to (-38.89, 43.33, 106.87) mm, rotated rx -180 ry 0 rz 180 deg; joints [-167.708, 65.216, -81.954, 167.182, 73.657, 3.663]
  MoveL 7157 to (-38.89, 43.33, 106.87) mm, rotated rx -180 ry 0 rz 180 deg; joints [-167.708, 65.216, -81.954, 167.182, 73.657, 3.663]
  Call Extruder(65.00093)
  MoveL 7158 to (-38.75, 43.06, 106.87) mm, rotated rx 180 ry 0 rz 180 deg; joints [-167.776, 65.201, -81.963, 167.251, 73.628, 3.649]
  MoveL 7159 to (-38.75, 43.06, 106.87) mm, rotated rx 180 ry 0 rz 180 deg; joints [-167.776, 65.201, -81.963, 167.251, 73.628, 3.649]
  Call Extruder(65.20748)
  MoveL 7160 to (-38.57, 42.75, 106.87) mm, rotated rx -180 ry 0 rz -180 deg; joints [-167.849, 65.182, -81.975, 167.325, 73.595, 3.634]
  MoveL 7161 to (-38.57, 42.75, 106.87) mm, rotated rx -180 ry 0 rz -180 deg; joints [-167.849, 65.182, -81.975, 167.325, 73.595, 3.634]
  Call Extruder(65.41482)
  MoveL 7162 to (-38.4, 42.45, 106.87) mm, rotated rx -180 ry 0 rz -180 deg; joints [-167.923, 65.164, -81.986, 167.4, 73.561, 3.619]
  MoveL 7163 to (-38.4, 42.45, 106.87) mm, rotated rx -180 ry 0 rz -180 deg; joints [-167.923, 65.164, -81.986, 167.4, 73.561, 3.619]
  Call Extruder(65.62293)
  MoveL 7164 to (-38.22, 42.15, 106.87) mm, rotated rx 180 ry 0 rz 180 deg; joints [-167.997, 65.146, -81.997, 167.475, 73.528, 3.604]
  MoveL 7165 to (-38.22, 42.15, 106.87) mm, rotated rx 180 ry 0 rz 180 deg; joints [-167.997, 65.146, -81.997, 167.475, 73.528, 3.604]
  Call Extruder(65.74065)
  MoveL 7166 to (-38.12, 41.98, 106.87) mm, rotated rx -180 ry 0 rz 180 deg; joints [-168.038, 65.136, -82.004, 167.517, 73.509, 3.596]
  MoveL 7167 to (-38.12, 41.98, 106.87) mm, rotated rx -180 ry 0 rz 180 deg; joints [-168.038, 65.136, -82.004, 167.517, 73.509, 3.596]
  Call Extruder(66.07349)
  MoveL 7168 to (-37.8, 41.52, 106.87) mm, rotated rx -180 ry 0 rz -180 deg; joints [-168.144, 65.104, -82.024, 167.624, 73.451, 3.576]
  MoveL 7169 to (-37.8, 41.52, 106.87) mm, rotated rx -180 ry 0 rz -180 deg; joints [-168.144, 65.104, -82.024, 167.624, 73.451, 3.576]
  Call Extruder(66.40752)
  MoveL 7170 to (-37.47, 41.07, 106.87) mm, rotated rx -180 ry 0 rz 180 deg; joints [-168.25, 65.072, -82.044, 167.731, 73.394, 3.556]
  MoveL 7171 to (-37.47, 41.07, 106.87) mm, rotated rx -180 ry 0 rz 180 deg; joints [-168.25, 65.072, -82.044, 167.731, 73.394, 3.556]
  Call Extruder(66.57511)
  MoveL 7172 to (-37.3, 40.85, 106.87) mm, rotated rx -180 ry 0 rz -180 deg; joints [-168.304, 65.056, -82.054, 167.785, 73.365, 3.546]
  Call Extruder(67.40442)
  MoveL 7173 to (-36.39, 39.81, 106.87) mm, rotated rx -180 ry 0 rz 180 deg; joints [-168.541, 64.97, -82.106, 168.024, 73.215, 3.505]
  Call Extruder(68.03549)
  MoveL 7174 to (-35.61, 39.11, 106.87) mm, rotated rx -180 ry 0 rz -180 deg; joints [-168.693, 64.899, -82.149, 168.175, 73.095, 3.484]
  MoveL 7175 to (-35.61, 39.11, 106.87) mm, rotated rx -180 ry 0 rz -180 deg; joints [-168.693, 64.899, -82.149, 168.175, 73.095, 3.484]
  Call Extruder(68.23306)
  MoveL 7176 to (-35.35, 38.9, 106.87) mm, rotated rx 180 ry 0 rz 180 deg; joints [-168.739, 64.877, -82.163, 168.221, 73.056, 3.478]
  Call Extruder(68.56708)
  MoveL 7177 to (-34.9, 38.57, 106.87) mm, rotated rx -180 ry 0 rz -180 deg; joints [-168.806, 64.837, -82.187, 168.287, 72.99, 3.471]
  MoveL 7178 to (-34.9, 38.57, 106.87) mm, rotated rx -180 ry 0 rz -180 deg; joints [-168.806, 64.837, -82.187, 168.287, 72.99, 3.471]
  Call Extruder(68.89991)
  MoveL 7179 to (-34.45, 38.24, 106.87) mm, rotated rx -180 ry 0 rz -180 deg; joints [-168.874, 64.797, -82.211, 168.354, 72.924, 3.463]
  MoveL 7180 to (-34.45, 38.24, 106.87) mm, rotated rx -180 ry 0 rz -180 deg; joints [-168.874, 64.797, -82.211, 168.354, 72.924, 3.463]
  Call Extruder(69.07916)
  MoveL 7181 to (-34.21, 38.06, 106.87) mm, rotated rx -180 ry 0 rz 180 deg; joints [-168.91, 64.775, -82.223, 168.39, 72.888, 3.46]
  MoveL 7182 to (-34.21, 38.06, 106.87) mm, rotated rx -180 ry 0 rz 180 deg; joints [-168.91, 64.775, -82.223, 168.39, 72.888, 3.46]
  Call Extruder(69.28727)
  MoveL 7183 to (-33.9, 37.89, 106.87) mm, rotated rx -180 ry 0 rz 180 deg; joints [-168.944, 64.749, -82.239, 168.422, 72.845, 3.458]
  MoveL 7184 to (-33.9, 37.89, 106.87) mm, rotated rx -180 ry 0 rz 180 deg; joints [-168.944, 64.749, -82.239, 168.422, 72.845, 3.458]
  Call Extruder(69.49460)
  MoveL 7185 to (-33.6, 37.71, 106.87) mm, rotated rx 180 ry 0 rz -180 deg; joints [-168.977, 64.723, -82.254, 168.454, 72.802, 3.457]
  MoveL 7186 to (-33.6, 37.71, 106.87) mm, rotated rx 180 ry 0 rz -180 deg; joints [-168.977, 64.723, -82.254, 168.454, 72.802, 3.457]
  Call Extruder(69.70115)
  MoveL 7187 to (-33.29, 37.54, 106.87) mm, rotated rx -180 ry 0 rz 180 deg; joints [-169.01, 64.697, -82.27, 168.486, 72.76, 3.455]
  MoveL 7188 to (-33.29, 37.54, 106.87) mm, rotated rx -180 ry 0 rz 180 deg; joints [-169.01, 64.697, -82.27, 168.486, 72.76, 3.455]
  Call Extruder(69.90692)
  MoveL 7189 to (-32.99, 37.36, 106.87) mm, rotated rx 180 ry 0 rz -180 deg; joints [-169.043, 64.671, -82.285, 168.518, 72.717, 3.453]
  MoveL 7190 to (-32.99, 37.36, 106.87) mm, rotated rx 180 ry 0 rz -180 deg; joints [-169.043, 64.671, -82.285, 168.518, 72.717, 3.453]
  Call Extruder(70.06523)
  MoveL 7191 to (-32.74, 37.26, 106.87) mm, rotated rx -180 ry 0 rz 180 deg; joints [-169.06, 64.65, -82.297, 168.534, 72.683, 3.455]
  MoveL 7192 to (-32.74, 37.26, 106.87) mm, rotated rx -180 ry 0 rz 180 deg; joints [-169.06, 64.65, -82.297, 168.534, 72.683, 3.455]
  Call Extruder(70.22293)
  MoveL 7193 to (-32.49, 37.15, 106.87) mm, rotated rx -180 ry 0 rz 180 deg; joints [-169.077, 64.629, -82.31, 168.549, 72.65, 3.457]
  MoveL 7194 to (-32.49, 37.15, 106.87) mm, rotated rx -180 ry 0 rz 180 deg; joints [-169.077, 64.629, -82.31, 168.549, 72.65, 3.457]
  Call Extruder(70.39301)
  MoveL 7195 to (-32.22, 37.04, 106.87) mm, rotated rx 180 ry 0 rz 180 deg; joints [-169.095, 64.606, -82.323, 168.566, 72.614, 3.459]
  MoveL 7196 to (-32.22, 37.04, 106.87) mm, rotated rx 180 ry 0 rz 180 deg; joints [-169.095, 64.606, -82.323, 168.566, 72.614, 3.459]
  Call Extruder(70.57535)
  MoveL 7197 to (-31.93, 36.91, 106.87) mm, rotated rx -180 ry 0 rz 180 deg; joints [-169.113, 64.581, -82.337, 168.583, 72.574, 3.461]
  MoveL 7198 to (-31.93, 36.91, 106.87) mm, rotated rx -180 ry 0 rz 180 deg; joints [-169.113, 64.581, -82.337, 168.583, 72.574, 3.461]
  Call Extruder(70.75692)
  MoveL 7199 to (-31.64, 36.79, 106.87) mm, rotated rx -180 ry 0 rz 180 deg; joints [-169.132, 64.557, -82.351, 168.6, 72.535, 3.463]
  MoveL 7200 to (-31.64, 36.79, 106.87) mm, rotated rx -180 ry 0 rz 180 deg; joints [-169.132, 64.557, -82.351, 168.6, 72.535, 3.463]
  Call Extruder(70.87038)
  MoveL 7201 to (-31.45, 36.73, 106.87) mm, rotated rx -180 ry 0 rz 180 deg; joints [-169.139, 64.541, -82.36, 168.606, 72.511, 3.466]
  MoveL 7202 to (-31.45, 36.73, 106.87) mm, rotated rx -180 ry 0 rz 180 deg; joints [-169.139, 64.541, -82.36, 168.606, 72.511, 3.466]
  Call Extruder(70.98339)
  MoveL 7203 to (-31.26, 36.67, 106.87) mm, rotated rx -180 ry 0 rz -180 deg; joints [-169.146, 64.525, -82.369, 168.612, 72.486, 3.469]
  MoveL 7204 to (-31.26, 36.67, 106.87) mm, rotated rx -180 ry 0 rz -180 deg; joints [-169.146, 64.525, -82.369, 168.612, 72.486, 3.469]
  Call Extruder(71.09596)
  MoveL 7205 to (-31.07, 36.61, 106.87) mm, rotated rx -180 ry 0 rz -180 deg; joints [-169.154, 64.51, -82.378, 168.618, 72.462, 3.471]
  MoveL 7206 to (-31.07, 36.61, 106.87) mm, rotated rx -180 ry 0 rz -180 deg; joints [-169.154, 64.51, -82.378, 168.618, 72.462, 3.471]
  Call Extruder(71.20809)
  MoveL 7207 to (-30.88, 36.55, 106.87) mm, rotated rx 180 ry 0 rz 180 deg; joints [-169.161, 64.494, -82.387, 168.624, 72.437, 3.474]
  MoveL 7208 to (-30.88, 36.55, 106.87) mm, rotated rx 180 ry 0 rz 180 deg; joints [-169.161, 64.494, -82.387, 168.624, 72.437, 3.474]
  Call Extruder(71.31977)
  MoveL 7209 to (-30.7, 36.49, 106.87) mm, rotated rx -180 ry 0 rz -180 deg; joints [-169.168, 64.478, -82.396, 168.63, 72.413, 3.477]
  MoveL 7210 to (-30.7, 36.49, 106.87) mm, rotated rx -180 ry 0 rz -180 deg; joints [-169.168, 64.478, -82.396, 168.63, 72.413, 3.477]
  Call Extruder(71.45084)
  MoveL 7211 to (-30.47, 36.42, 106.87) mm, rotated rx -180 ry 0 rz 180 deg; joints [-169.175, 64.46, -82.406, 168.636, 72.384, 3.481]
  MoveL 7212 to (-30.47, 36.42, 106.87) mm, rotated rx -180 ry 0 rz 180 deg; joints [-169.175, 64.46, -82.406, 168.636, 72.384, 3.481]
  Call Extruder(71.58135)
  MoveL 7213 to (-30.25, 36.35, 106.87) mm, rotated rx -180 ry 0 rz -180 deg; joints [-169.182, 64.441, -82.417, 168.641, 72.355, 3.485]
  MoveL 7214 to (-30.25, 36.35, 106.87) mm, rotated rx -180 ry 0 rz -180 deg; joints [-169.182, 64.441, -82.417, 168.641, 72.355, 3.485]
  Call Extruder(71.71129)
  MoveL 7215 to (-30.02, 36.28, 106.87) mm, rotated rx -180 ry 0 rz -180 deg; joints [-169.19, 64.423, -82.427, 168.647, 72.326, 3.488]
  MoveL 7216 to (-30.02, 36.28, 106.87) mm, rotated rx -180 ry 0 rz -180 deg; joints [-169.19, 64.423, -82.427, 168.647, 72.326, 3.488]
  Call Extruder(71.84067)
  MoveL 7217 to (-29.8, 36.22, 106.87) mm, rotated rx -180 ry 0 rz -180 deg; joints [-169.197, 64.404, -82.438, 168.653, 72.297, 3.492]
  MoveL 7218 to (-29.8, 36.22, 106.87) mm, rotated rx -180 ry 0 rz -180 deg; joints [-169.197, 64.404, -82.438, 168.653, 72.297, 3.492]
  Call Extruder(71.96263)
  MoveL 7219 to (-29.59, 36.16, 106.87) mm, rotated rx 180 ry 0 rz 180 deg; joints [-169.202, 64.386, -82.447, 168.656, 72.269, 3.496]
  MoveL 7220 to (-29.59, 36.16, 106.87) mm, rotated rx 180 ry 0 rz 180 deg; joints [-169.202, 64.386, -82.447, 168.656, 72.269, 3.496]
  Call Extruder(72.07748)
  MoveL 7221 to (-29.38, 36.12, 106.87) mm, rotated rx 180 ry 0 rz 180 deg; joints [-169.203, 64.37, -82.457, 168.656, 72.244, 3.501]
  MoveL 7222 to (-29.38, 36.12, 106.87) mm, rotated rx 180 ry 0 rz 180 deg; joints [-169.203, 64.37, -82.457, 168.656, 72.244, 3.501]
  Call Extruder(72.19188)
  MoveL 7223 to (-29.18, 36.07, 106.87) mm, rotated rx -180 ry 0 rz 180 deg; joints [-169.205, 64.353, -82.466, 168.656, 72.218, 3.506]
  MoveL 7224 to (-29.18, 36.07, 106.87) mm, rotated rx -180 ry 0 rz 180 deg; joints [-169.205, 64.353, -82.466, 168.656, 72.218, 3.506]
  Call Extruder(72.30582)
  MoveL 7225 to (-28.97, 36.03, 106.87) mm, rotated rx -180 ry 0 rz -180 deg; joints [-169.207, 64.336, -82.475, 168.656, 72.192, 3.511]
  MoveL 7226 to (-28.97, 36.03, 106.87) mm, rotated rx -180 ry 0 rz -180 deg; joints [-169.207, 64.336, -82.475, 168.656, 72.192, 3.511]
  Call Extruder(72.41931)
  MoveL 7227 to (-28.77, 35.98, 106.87) mm, rotated rx 180 ry 0 rz 180 deg; joints [-169.208, 64.319, -82.485, 168.656, 72.167, 3.516]
  MoveL 7228 to (-28.77, 35.98, 106.87) mm, rotated rx 180 ry 0 rz 180 deg; joints [-169.208, 64.319, -82.485, 168.656, 72.167, 3.516]
  Call Extruder(72.55659)
  MoveL 7229 to (-28.52, 35.93, 106.87) mm, rotated rx -180 ry 0 rz -180 deg; joints [-169.209, 64.299, -82.496, 168.655, 72.135, 3.522]
  MoveL 7230 to (-28.52, 35.93, 106.87) mm, rotated rx -180 ry 0 rz -180 deg; joints [-169.209, 64.299, -82.496, 168.655, 72.135, 3.522]
  Call Extruder(72.69326)
  MoveL 7231 to (-28.27, 35.88, 106.87) mm, rotated rx -180 ry 0 rz -180 deg; joints [-169.209, 64.278, -82.507, 168.654, 72.104, 3.528]
  MoveL 7232 to (-28.27, 35.88, 106.87) mm, rotated rx -180 ry 0 rz -180 deg; joints [-169.209, 64.278, -82.507, 168.654, 72.104, 3.528]
  Call Extruder(72.82933)
  MoveL 7233 to (-28.02, 35.83, 106.87) mm, rotated rx -180 ry 0 rz 180 deg; joints [-169.21, 64.258, -82.519, 168.652, 72.073, 3.535]
  MoveL 7234 to (-28.02, 35.83, 106.87) mm, rotated rx -180 ry 0 rz 180 deg; joints [-169.21, 64.258, -82.519, 168.652, 72.073, 3.535]
  Call Extruder(72.96478)
  MoveL 7235 to (-27.77, 35.78, 106.87) mm, rotated rx 180 ry 0 rz 180 deg; joints [-169.21, 64.237, -82.53, 168.651, 72.042, 3.541]
  MoveL 7236 to (-27.77, 35.78, 106.87) mm, rotated rx 180 ry 0 rz 180 deg; joints [-169.21, 64.237, -82.53, 168.651, 72.042, 3.541]
  Call Extruder(73.09962)
  MoveL 7237 to (-27.52, 35.73, 106.87) mm, rotated rx -180 ry 0 rz 180 deg; joints [-169.211, 64.217, -82.541, 168.65, 72.011, 3.547]
  MoveL 7238 to (-27.52, 35.73, 106.87) mm, rotated rx -180 ry 0 rz 180 deg; joints [-169.211, 64.217, -82.541, 168.65, 72.011, 3.547]
  Call Extruder(73.23385)
  MoveL 7239 to (-27.28, 35.68, 106.87) mm, rotated rx 180 ry 0 rz 180 deg; joints [-169.212, 64.196, -82.552, 168.648, 71.98, 3.554]
  MoveL 7240 to (-27.28, 35.68, 106.87) mm, rotated rx 180 ry 0 rz 180 deg; joints [-169.212, 64.196, -82.552, 168.648, 71.98, 3.554]
  Call Extruder(73.36747)
  MoveL 7241 to (-27.03, 35.63, 106.87) mm, rotated rx 180 ry 0 rz 180 deg; joints [-169.212, 64.176, -82.563, 168.647, 71.949, 3.56]
  MoveL 7242 to (-27.03, 35.63, 106.87) mm, rotated rx 180 ry 0 rz 180 deg; joints [-169.212, 64.176, -82.563, 168.647, 71.949, 3.56]
  Call Extruder(73.52957)
  MoveL 7243 to (-26.72, 35.59, 106.87) mm, rotated rx -180 ry 0 rz 180 deg; joints [-169.21, 64.151, -82.577, 168.641, 71.911, 3.569]
  MoveL 7244 to (-26.72, 35.59, 106.87) mm, rotated rx -180 ry 0 rz 180 deg; joints [-169.21, 64.151, -82.577, 168.641, 71.911, 3.569]
  Call Extruder(73.69094)
  MoveL 7245 to (-26.41, 35.54, 106.87) mm, rotated rx 180 ry 0 rz 180 deg; joints [-169.207, 64.126, -82.59, 168.636, 71.873, 3.578]
  MoveL 7246 to (-26.41, 35.54, 106.87) mm, rotated rx 180 ry 0 rz 180 deg; joints [-169.207, 64.126, -82.59, 168.636, 71.873, 3.578]
  Call Extruder(73.85158)
  MoveL 7247 to (-26.11, 35.49, 106.87) mm, rotated rx -180 ry 0 rz -180 deg; joints [-169.204, 64.1, -82.604, 168.63, 71.836, 3.587]
  MoveL 7248 to (-26.11, 35.49, 106.87) mm, rotated rx -180 ry 0 rz -180 deg; joints [-169.204, 64.1, -82.604, 168.63, 71.836, 3.587]
  Call Extruder(74.01150)
  MoveL 7249 to (-25.8, 35.44, 106.87) mm, rotated rx -180 ry 0 rz 180 deg; joints [-169.201, 64.075, -82.617, 168.625, 71.798, 3.596]
  MoveL 7250 to (-25.8, 35.44, 106.87) mm, rotated rx -180 ry 0 rz 180 deg; joints [-169.201, 64.075, -82.617, 168.625, 71.798, 3.596]
  Call Extruder(74.17069)
  MoveL 7251 to (-25.5, 35.39, 106.87) mm, rotated rx 180 ry 0 rz -180 deg; joints [-169.198, 64.05, -82.631, 168.619, 71.76, 3.605]
  MoveL 7252 to (-25.5, 35.39, 106.87) mm, rotated rx 180 ry 0 rz -180 deg; joints [-169.198, 64.05, -82.631, 168.619, 71.76, 3.605]
  Call Extruder(74.32915)
  MoveL 7253 to (-25.19, 35.34, 106.87) mm, rotated rx -180 ry 0 rz -180 deg; joints [-169.195, 64.025, -82.644, 168.613, 71.723, 3.614]
  MoveL 7254 to (-25.19, 35.34, 106.87) mm, rotated rx -180 ry 0 rz -180 deg; joints [-169.195, 64.025, -82.644, 168.613, 71.723, 3.614]
  Call Extruder(74.52802)
  MoveL 7255 to (-24.8, 35.3, 106.87) mm, rotated rx 180 ry 0 rz 180 deg; joints [-169.187, 63.993, -82.661, 168.601, 71.676, 3.627]
  MoveL 7256 to (-24.8, 35.3, 106.87) mm, rotated rx 180 ry 0 rz 180 deg; joints [-169.187, 63.993, -82.661, 168.601, 71.676, 3.627]
  Call Extruder(74.72603)
  MoveL 7257 to (-24.42, 35.25, 106.87) mm, rotated rx -180 ry 0 rz -180 deg; joints [-169.178, 63.961, -82.677, 168.589, 71.629, 3.64]
  MoveL 7258 to (-24.42, 35.25, 106.87) mm, rotated rx -180 ry 0 rz -180 deg; joints [-169.178, 63.961, -82.677, 168.589, 71.629, 3.64]
  Call Extruder(74.92317)
  MoveL 7259 to (-24.03, 35.21, 106.87) mm, rotated rx 180 ry 0 rz 180 deg; joints [-169.17, 63.93, -82.694, 168.577, 71.582, 3.653]
  MoveL 7260 to (-24.03, 35.21, 106.87) mm, rotated rx 180 ry 0 rz 180 deg; joints [-169.17, 63.93, -82.694, 168.577, 71.582, 3.653]
  Call Extruder(75.11944)
  MoveL 7261 to (-23.64, 35.16, 106.87) mm, rotated rx -180 ry 0 rz 180 deg; joints [-169.161, 63.898, -82.711, 168.565, 71.535, 3.666]
  MoveL 7262 to (-23.64, 35.16, 106.87) mm, rotated rx -180 ry 0 rz 180 deg; joints [-169.161, 63.898, -82.711, 168.565, 71.535, 3.666]
  Call Extruder(75.36513)
  MoveL 7263 to (-23.15, 35.11, 106.87) mm, rotated rx -180 ry 0 rz 180 deg; joints [-169.147, 63.858, -82.731, 168.546, 71.476, 3.683]
  MoveL 7264 to (-23.15, 35.11, 106.87) mm, rotated rx -180 ry 0 rz 180 deg; joints [-169.147, 63.858, -82.731, 168.546, 71.476, 3.683]
  Call Extruder(75.65986)
  MoveL 7265 to (-22.56, 35.07, 106.87) mm, rotated rx -180 ry 0 rz -180 deg; joints [-169.127, 63.809, -82.756, 168.52, 71.406, 3.705]
  MoveL 7266 to (-22.56, 35.07, 106.87) mm, rotated rx -180 ry 0 rz -180 deg; joints [-169.127, 63.809, -82.756, 168.52, 71.406, 3.705]
  Call Extruder(75.95326)
  MoveL 7267 to (-21.97, 35.02, 106.87) mm, rotated rx 180 ry 0 rz 180 deg; joints [-169.107, 63.761, -82.781, 168.494, 71.335, 3.727]
  MoveL 7268 to (-21.97, 35.02, 106.87) mm, rotated rx 180 ry 0 rz 180 deg; joints [-169.107, 63.761, -82.781, 168.494, 71.335, 3.727]
  Call Extruder(76.38658)
  MoveL 7269 to (-21.1, 34.97, 106.87) mm, rotated rx -180 ry 0 rz -180 deg; joints [-169.069, 63.689, -82.817, 168.447, 71.232, 3.763]
  MoveL 7270 to (-21.1, 34.97, 106.87) mm, rotated rx -180 ry 0 rz -180 deg; joints [-169.069, 63.689, -82.817, 168.447, 71.232, 3.763]
  Call Extruder(76.95875)
  MoveL 7271 to (-19.94, 34.93, 106.87) mm, rotated rx 180 ry 0 rz -180 deg; joints [-169.014, 63.594, -82.865, 168.379, 71.096, 3.812]
  MoveL 7272 to (-19.94, 34.93, 106.87) mm, rotated rx 180 ry 0 rz -180 deg; joints [-169.014, 63.594, -82.865, 168.379, 71.096, 3.812]
  Call Extruder(77.38658)
  MoveL 7273 to (-19.06, 34.91, 106.87) mm, rotated rx -180 ry 0 rz -180 deg; joints [-168.967, 63.522, -82.9, 168.323, 70.994, 3.851]
  Call Extruder(194.03526)
  MoveL 7274 to (219.06, 34.91, 106.87) mm, rotated rx -180 ry 0 rz 180 deg; joints [-30.588, 52.278, -85.09, 35.119, 117.806, 18.164]
  MoveL 7275 to (219.06, 34.91, 106.87) mm, rotated rx -180 ry 0 rz 180 deg; joints [-30.588, 52.278, -85.09, 35.119, 117.806, 18.164]
  Call Extruder(194.75084)
  MoveL 7276 to (220.52, 34.95, 106.87) mm, rotated rx -180 ry 0 rz 180 deg; joints [-30.009, 52.422, -85.093, 34.454, 117.869, 17.782]
  MoveL 7277 to (220.52, 34.95, 106.87) mm, rotated rx -180 ry 0 rz 180 deg; joints [-30.009, 52.422, -85.093, 34.454, 117.869, 17.782]
  Call Extruder(195.32557)
  MoveL 7278 to (221.68, 35, 106.87) mm, rotated rx 180 ry 0 rz 180 deg; joints [-29.572, 52.538, -85.095, 33.949, 117.907, 17.489]
  MoveL 7279 to (221.68, 35, 106.87) mm, rotated rx 180 ry 0 rz 180 deg; joints [-29.572, 52.538, -85.095, 33.949, 117.907, 17.489]
  Call Extruder(195.61897)
  MoveL 7280 to (222.27, 35.05, 106.87) mm, rotated rx -180 ry 0 rz 180 deg; joints [-29.371, 52.598, -85.096, 33.715, 117.918, 17.35]
  MoveL 7281 to (222.27, 35.05, 106.87) mm, rotated rx -180 ry 0 rz 180 deg; joints [-29.371, 52.598, -85.096, 33.715, 117.918, 17.35]
  Call Extruder(195.91369)
  MoveL 7282 to (222.86, 35.09, 106.87) mm, rotated rx -180 ry 0 rz 180 deg; joints [-29.173, 52.658, -85.096, 33.483, 117.927, 17.213]
  MoveL 7283 to (222.86, 35.09, 106.87) mm, rotated rx -180 ry 0 rz 180 deg; joints [-29.173, 52.658, -85.096, 33.483, 117.927, 17.213]
  Call Extruder(196.20975)
  MoveL 7284 to (223.45, 35.14, 106.87) mm, rotated rx -180 ry 0 rz 180 deg; joints [-28.978, 52.718, -85.097, 33.255, 117.935, 17.077]
  MoveL 7285 to (223.45, 35.14, 106.87) mm, rotated rx -180 ry 0 rz 180 deg; joints [-28.978, 52.718, -85.097, 33.255, 117.935, 17.077]
  Call Extruder(196.40602)
  MoveL 7286 to (223.84, 35.18, 106.87) mm, rotated rx -180 ry 0 rz 180 deg; joints [-28.862, 52.758, -85.097, 33.118, 117.936, 16.993]
  MoveL 7287 to (223.84, 35.18, 106.87) mm, rotated rx -180 ry 0 rz 180 deg; joints [-28.862, 52.758, -85.097, 33.118, 117.936, 16.993]
  Call Extruder(196.60317)
  MoveL 7288 to (224.22, 35.23, 106.87) mm, rotated rx -180 ry 0 rz 180 deg; joints [-28.747, 52.799, -85.097, 32.982, 117.935, 16.91]
  MoveL 7289 to (224.22, 35.23, 106.87) mm, rotated rx -180 ry 0 rz 180 deg; joints [-28.747, 52.799, -85.097, 32.982, 117.935, 16.91]
  Call Extruder(196.80118)
  MoveL 7290 to (224.61, 35.28, 106.87) mm, rotated rx 180 ry 0 rz 180 deg; joints [-28.633, 52.839, -85.098, 32.847, 117.935, 16.828]
  MoveL 7291 to (224.61, 35.28, 106.87) mm, rotated rx 180 ry 0 rz 180 deg; joints [-28.633, 52.839, -85.098, 32.847, 117.935, 16.828]
  Call Extruder(197.00005)
  MoveL 7292 to (225, 35.32, 106.87) mm, rotated rx 180 ry 0 rz 180 deg; joints [-28.52, 52.88, -85.098, 32.713, 117.933, 16.746]
  MoveL 7293 to (225, 35.32, 106.87) mm, rotated rx 180 ry 0 rz 180 deg; joints [-28.52, 52.88, -85.098, 32.713, 117.933, 16.746]
  Call Extruder(197.17913)
  MoveL 7294 to (225.34, 35.37, 106.87) mm, rotated rx -180 ry 0 rz -180 deg; joints [-28.425, 52.916, -85.098, 32.599, 117.93, 16.675]
  MoveL 7295 to (225.34, 35.37, 106.87) mm, rotated rx -180 ry 0 rz -180 deg; joints [-28.425, 52.916, -85.098, 32.599, 117.93, 16.675]
  Call Extruder(197.33831)
  MoveL 7296 to (225.65, 35.42, 106.87) mm, rotated rx 180 ry 0 rz 180 deg; joints [-28.346, 52.949, -85.098, 32.505, 117.925, 16.616]
  MoveL 7297 to (225.65, 35.42, 106.87) mm, rotated rx 180 ry 0 rz 180 deg; joints [-28.346, 52.949, -85.098, 32.505, 117.925, 16.616]
  Call Extruder(197.49823)
  MoveL 7298 to (225.96, 35.47, 106.87) mm, rotated rx 180 ry 0 rz 180 deg; joints [-28.267, 52.981, -85.098, 32.41, 117.921, 16.556]
  MoveL 7299 to (225.96, 35.47, 106.87) mm, rotated rx 180 ry 0 rz 180 deg; joints [-28.267, 52.981, -85.098, 32.41, 117.921, 16.556]
  Call Extruder(197.65886)
  MoveL 7300 to (226.26, 35.51, 106.87) mm, rotated rx -180 ry 0 rz 180 deg; joints [-28.19, 53.014, -85.098, 32.317, 117.915, 16.497]
  MoveL 7301 to (226.26, 35.51, 106.87) mm, rotated rx -180 ry 0 rz 180 deg; joints [-28.19, 53.014, -85.098, 32.317, 117.915, 16.497]
  Call Extruder(197.82023)
  MoveL 7302 to (226.57, 35.56, 106.87) mm, rotated rx -180 ry 0 rz 180 deg; joints [-28.112, 53.046, -85.098, 32.224, 117.91, 16.438]
  MoveL 7303 to (226.57, 35.56, 106.87) mm, rotated rx -180 ry 0 rz 180 deg; joints [-28.112, 53.046, -85.098, 32.224, 117.91, 16.438]
  Call Extruder(197.98233)
  MoveL 7304 to (226.87, 35.61, 106.87) mm, rotated rx -180 ry 0 rz 180 deg; joints [-28.036, 53.079, -85.098, 32.131, 117.903, 16.379]
  MoveL 7305 to (226.87, 35.61, 106.87) mm, rotated rx -180 ry 0 rz 180 deg; joints [-28.036, 53.079, -85.098, 32.131, 117.903, 16.379]
  Call Extruder(198.13052)
  MoveL 7306 to (227.15, 35.66, 106.87) mm, rotated rx -180 ry 0 rz -180 deg; joints [-27.971, 53.109, -85.098, 32.052, 117.897, 16.328]
  MoveL 7307 to (227.15, 35.66, 106.87) mm, rotated rx -180 ry 0 rz -180 deg; joints [-27.971, 53.109, -85.098, 32.052, 117.897, 16.328]
  Call Extruder(198.26476)
  MoveL 7308 to (227.4, 35.71, 106.87) mm, rotated rx -180 ry 0 rz 180 deg; joints [-27.915, 53.136, -85.098, 31.984, 117.889, 16.284]
  MoveL 7309 to (227.4, 35.71, 106.87) mm, rotated rx -180 ry 0 rz 180 deg; joints [-27.915, 53.136, -85.098, 31.984, 117.889, 16.284]
  Call Extruder(198.39960)
  MoveL 7310 to (227.65, 35.76, 106.87) mm, rotated rx 180 ry 0 rz 180 deg; joints [-27.861, 53.163, -85.098, 31.918, 117.881, 16.24]
  MoveL 7311 to (227.65, 35.76, 106.87) mm, rotated rx 180 ry 0 rz 180 deg; joints [-27.861, 53.163, -85.098, 31.918, 117.881, 16.24]
  Call Extruder(198.53505)
  MoveL 7312 to (227.9, 35.81, 106.87) mm, rotated rx 180 ry 0 rz 180 deg; joints [-27.807, 53.189, -85.097, 31.851, 117.874, 16.196]
  MoveL 7313 to (227.9, 35.81, 106.87) mm, rotated rx 180 ry 0 rz 180 deg; joints [-27.807, 53.189, -85.097, 31.851, 117.874, 16.196]
  Call Extruder(198.67111)
  MoveL 7314 to (228.15, 35.86, 106.87) mm, rotated rx 180 ry 0 rz 180 deg; joints [-27.753, 53.216, -85.097, 31.785, 117.865, 16.153]
  MoveL 7315 to (228.15, 35.86, 106.87) mm, rotated rx 180 ry 0 rz 180 deg; joints [-27.753, 53.216, -85.097, 31.785, 117.865, 16.153]
  Call Extruder(198.80779)
  MoveL 7316 to (228.4, 35.91, 106.87) mm, rotated rx 180 ry 0 rz 180 deg; joints [-27.699, 53.244, -85.097, 31.719, 117.857, 16.109]
  MoveL 7317 to (228.4, 35.91, 106.87) mm, rotated rx 180 ry 0 rz 180 deg; joints [-27.699, 53.244, -85.097, 31.719, 117.857, 16.109]
  Call Extruder(198.94507)
  MoveL 7318 to (228.64, 35.96, 106.87) mm, rotated rx -180 ry 0 rz 180 deg; joints [-27.646, 53.271, -85.097, 31.654, 117.849, 16.066]
  MoveL 7319 to (228.64, 35.96, 106.87) mm, rotated rx -180 ry 0 rz 180 deg; joints [-27.646, 53.271, -85.097, 31.654, 117.849, 16.066]
  Call Extruder(199.07074)
  MoveL 7320 to (228.87, 36, 106.87) mm, rotated rx -180 ry 0 rz 180 deg; joints [-27.599, 53.295, -85.097, 31.596, 117.841, 16.028]
  MoveL 7321 to (228.87, 36, 106.87) mm, rotated rx -180 ry 0 rz 180 deg; joints [-27.599, 53.295, -85.097, 31.596, 117.841, 16.028]
  Call Extruder(199.18469)
  MoveL 7322 to (229.08, 36.05, 106.87) mm, rotated rx 180 ry 0 rz 180 deg; joints [-27.559, 53.318, -85.096, 31.546, 117.832, 15.994]
  MoveL 7323 to (229.08, 36.05, 106.87) mm, rotated rx 180 ry 0 rz 180 deg; joints [-27.559, 53.318, -85.096, 31.546, 117.832, 15.994]
  Call Extruder(199.29909)
  MoveL 7324 to (229.28, 36.09, 106.87) mm, rotated rx -180 ry 0 rz 180 deg; joints [-27.518, 53.34, -85.096, 31.496, 117.824, 15.96]
  MoveL 7325 to (229.28, 36.09, 106.87) mm, rotated rx -180 ry 0 rz 180 deg; joints [-27.518, 53.34, -85.096, 31.496, 117.824, 15.96]
  Call Extruder(199.41394)
  MoveL 7326 to (229.48, 36.14, 106.87) mm, rotated rx 180 ry 0 rz 180 deg; joints [-27.479, 53.362, -85.096, 31.446, 117.816, 15.926]
  MoveL 7327 to (229.48, 36.14, 106.87) mm, rotated rx 180 ry 0 rz 180 deg; joints [-27.479, 53.362, -85.096, 31.446, 117.816, 15.926]
  Call Extruder(199.52925)
  MoveL 7328 to (229.69, 36.18, 106.87) mm, rotated rx -180 ry 0 rz 180 deg; joints [-27.439, 53.384, -85.096, 31.397, 117.808, 15.893]
  MoveL 7329 to (229.69, 36.18, 106.87) mm, rotated rx -180 ry 0 rz 180 deg; joints [-27.439, 53.384, -85.096, 31.397, 117.808, 15.893]
  Call Extruder(199.65431)
  MoveL 7330 to (229.91, 36.25, 106.87) mm, rotated rx -180 ry 0 rz 180 deg; joints [-27.407, 53.409, -85.095, 31.355, 117.795, 15.862]
  MoveL 7331 to (229.91, 36.25, 106.87) mm, rotated rx -180 ry 0 rz 180 deg; joints [-27.407, 53.409, -85.095, 31.355, 117.795, 15.862]
  Call Extruder(199.77989)
  MoveL 7332 to (230.12, 36.31, 106.87) mm, rotated rx 180 ry 0 rz 180 deg; joints [-27.376, 53.433, -85.095, 31.315, 117.783, 15.832]
  MoveL 7333 to (230.12, 36.31, 106.87) mm, rotated rx 180 ry 0 rz 180 deg; joints [-27.376, 53.433, -85.095, 31.315, 117.783, 15.832]
  Call Extruder(199.90597)
  MoveL 7334 to (230.34, 36.37, 106.87) mm, rotated rx -180 ry 0 rz 180 deg; joints [-27.345, 53.458, -85.095, 31.274, 117.77, 15.801]
  MoveL 7335 to (230.34, 36.37, 106.87) mm, rotated rx -180 ry 0 rz 180 deg; joints [-27.345, 53.458, -85.095, 31.274, 117.77, 15.801]
  Call Extruder(200.01064)
  MoveL 7336 to (230.52, 36.43, 106.87) mm, rotated rx -180 ry 0 rz 180 deg; joints [-27.321, 53.478, -85.094, 31.243, 117.759, 15.777]
  MoveL 7337 to (230.52, 36.43, 106.87) mm, rotated rx -180 ry 0 rz 180 deg; joints [-27.321, 53.478, -85.094, 31.243, 117.759, 15.777]
  Call Extruder(200.11570)
  MoveL 7338 to (230.7, 36.49, 106.87) mm, rotated rx 180 ry 0 rz -180 deg; joints [-27.299, 53.499, -85.094, 31.213, 117.747, 15.754]
  MoveL 7339 to (230.7, 36.49, 106.87) mm, rotated rx 180 ry 0 rz -180 deg; joints [-27.299, 53.499, -85.094, 31.213, 117.747, 15.754]
  Call Extruder(200.22759)
  MoveL 7340 to (230.88, 36.55, 106.87) mm, rotated rx -180 ry 0 rz 180 deg; joints [-27.276, 53.52, -85.094, 31.182, 117.735, 15.73]
  MoveL 7341 to (230.88, 36.55, 106.87) mm, rotated rx -180 ry 0 rz 180 deg; joints [-27.276, 53.52, -85.094, 31.182, 117.735, 15.73]
  Call Extruder(200.33994)
  MoveL 7342 to (231.07, 36.61, 106.87) mm, rotated rx 180 ry 0 rz 180 deg; joints [-27.253, 53.542, -85.093, 31.151, 117.722, 15.705]
  MoveL 7343 to (231.07, 36.61, 106.87) mm, rotated rx 180 ry 0 rz 180 deg; joints [-27.253, 53.542, -85.093, 31.151, 117.722, 15.705]
  Call Extruder(200.45272)
  MoveL 7344 to (231.26, 36.67, 106.87) mm, rotated rx 180 ry 0 rz 180 deg; joints [-27.231, 53.563, -85.093, 31.121, 117.709, 15.681]
  MoveL 7345 to (231.26, 36.67, 106.87) mm, rotated rx 180 ry 0 rz 180 deg; joints [-27.231, 53.563, -85.093, 31.121, 117.709, 15.681]
  Call Extruder(200.56596)
  MoveL 7346 to (231.45, 36.73, 106.87) mm, rotated rx -180 ry 0 rz 180 deg; joints [-27.208, 53.585, -85.093, 31.09, 117.697, 15.657]
  MoveL 7347 to (231.45, 36.73, 106.87) mm, rotated rx -180 ry 0 rz 180 deg; joints [-27.208, 53.585, -85.093, 31.09, 117.697, 15.657]
  Call Extruder(200.67963)
  MoveL 7348 to (231.64, 36.79, 106.87) mm, rotated rx -180 ry 0 rz 180 deg; joints [-27.185, 53.606, -85.092, 31.06, 117.684, 15.632]
  MoveL 7349 to (231.64, 36.79, 106.87) mm, rotated rx -180 ry 0 rz 180 deg; joints [-27.185, 53.606, -85.092, 31.06, 117.684, 15.632]
  Call Extruder(200.86159)
  MoveL 7350 to (231.93, 36.91, 106.87) mm, rotated rx -180 ry 0 rz 180 deg; joints [-27.167, 53.641, -85.092, 31.03, 117.659, 15.603]
  MoveL 7351 to (231.93, 36.91, 106.87) mm, rotated rx -180 ry 0 rz 180 deg; joints [-27.167, 53.641, -85.092, 31.03, 117.659, 15.603]
  Call Extruder(201.04431)
  MoveL 7352 to (232.22, 37.04, 106.87) mm, rotated rx -180 ry 0 rz 180 deg; joints [-27.149, 53.675, -85.091, 31.001, 117.633, 15.573]
  MoveL 7353 to (232.22, 37.04, 106.87) mm, rotated rx -180 ry 0 rz 180 deg; joints [-27.149, 53.675, -85.091, 31.001, 117.633, 15.573]
  Call Extruder(201.21473)
  MoveL 7354 to (232.49, 37.15, 106.87) mm, rotated rx 180 ry 0 rz -180 deg; joints [-27.133, 53.708, -85.09, 30.975, 117.609, 15.546]
  MoveL 7355 to (232.49, 37.15, 106.87) mm, rotated rx 180 ry 0 rz -180 deg; joints [-27.133, 53.708, -85.09, 30.975, 117.609, 15.546]
  Call Extruder(201.37273)
  MoveL 7356 to (232.74, 37.26, 106.87) mm, rotated rx -180 ry 0 rz 180 deg; joints [-27.121, 53.737, -85.089, 30.953, 117.587, 15.522]
  MoveL 7357 to (232.74, 37.26, 106.87) mm, rotated rx -180 ry 0 rz 180 deg; joints [-27.121, 53.737, -85.089, 30.953, 117.587, 15.522]
  Call Extruder(201.53133)
  MoveL 7358 to (232.99, 37.36, 106.87) mm, rotated rx -180 ry 0 rz 180 deg; joints [-27.108, 53.767, -85.089, 30.931, 117.564, 15.498]
  MoveL 7359 to (232.99, 37.36, 106.87) mm, rotated rx -180 ry 0 rz 180 deg; joints [-27.108, 53.767, -85.089, 30.931, 117.564, 15.498]
  Call Extruder(201.73750)
  MoveL 7360 to (233.29, 37.54, 106.87) mm, rotated rx -180 ry 0 rz 180 deg; joints [-27.12, 53.805, -85.088, 30.933, 117.527, 15.481]
  MoveL 7361 to (233.29, 37.54, 106.87) mm, rotated rx -180 ry 0 rz 180 deg; joints [-27.12, 53.805, -85.088, 30.933, 117.527, 15.481]
  Call Extruder(201.94444)
  MoveL 7362 to (233.6, 37.71, 106.87) mm, rotated rx -180 ry 0 rz -180 deg; joints [-27.132, 53.844, -85.087, 30.936, 117.49, 15.464]
  MoveL 7363 to (233.6, 37.71, 106.87) mm, rotated rx -180 ry 0 rz -180 deg; joints [-27.132, 53.844, -85.087, 30.936, 117.49, 15.464]
  Call Extruder(202.15217)
  MoveL 7364 to (233.9, 37.89, 106.87) mm, rotated rx -180 ry 0 rz 180 deg; joints [-27.144, 53.882, -85.086, 30.939, 117.453, 15.447]
  MoveL 7365 to (233.9, 37.89, 106.87) mm, rotated rx -180 ry 0 rz 180 deg; joints [-27.144, 53.882, -85.086, 30.939, 117.453, 15.447]
  Call Extruder(202.36067)
  MoveL 7366 to (234.21, 38.06, 106.87) mm, rotated rx -180 ry 0 rz 180 deg; joints [-27.156, 53.921, -85.085, 30.942, 117.416, 15.431]
  MoveL 7367 to (234.21, 38.06, 106.87) mm, rotated rx -180 ry 0 rz 180 deg; joints [-27.156, 53.921, -85.085, 30.942, 117.416, 15.431]
  Call Extruder(202.54021)
  MoveL 7368 to (234.45, 38.24, 106.87) mm, rotated rx 180 ry 0 rz -180 deg; joints [-27.187, 53.953, -85.084, 30.966, 117.379, 15.427]
  MoveL 7369 to (234.45, 38.24, 106.87) mm, rotated rx 180 ry 0 rz -180 deg; joints [-27.187, 53.953, -85.084, 30.966, 117.379, 15.427]
  Call Extruder(202.87363)
  MoveL 7370 to (234.9, 38.57, 106.87) mm, rotated rx 180 ry 0 rz 180 deg; joints [-27.245, 54.014, -85.082, 31.013, 117.31, 15.42]
  MoveL 7371 to (234.9, 38.57, 106.87) mm, rotated rx 180 ry 0 rz 180 deg; joints [-27.245, 54.014, -85.082, 31.013, 117.31, 15.42]
  Call Extruder(203.20823)
  MoveL 7372 to (235.35, 38.9, 106.87) mm, rotated rx 180 ry 0 rz 180 deg; joints [-27.302, 54.074, -85.08, 31.058, 117.241, 15.412]
  Call Extruder(204.03618)
  MoveL 7373 to (236.39, 39.81, 106.87) mm, rotated rx -180 ry 0 rz 180 deg; joints [-27.525, 54.22, -85.074, 31.259, 117.053, 15.434]
  Call Extruder(204.86412)
  MoveL 7374 to (237.3, 40.85, 106.87) mm, rotated rx 180 ry 0 rz 180 deg; joints [-27.851, 54.36, -85.069, 31.573, 116.841, 15.509]
  Call Extruder(205.03142)
  MoveL 7375 to (237.47, 41.07, 106.87) mm, rotated rx -180 ry 0 rz 180 deg; joints [-27.932, 54.387, -85.067, 31.653, 116.795, 15.531]
  MoveL 7376 to (237.47, 41.07, 106.87) mm, rotated rx -180 ry 0 rz 180 deg; joints [-27.932, 54.387, -85.067, 31.653, 116.795, 15.531]
  Call Extruder(205.36483)
  MoveL 7377 to (237.79, 41.52, 106.87) mm, rotated rx -180 ry 0 rz 180 deg; joints [-28.091, 54.441, -85.065, 31.809, 116.704, 15.575]
  MoveL 7378 to (237.79, 41.52, 106.87) mm, rotated rx -180 ry 0 rz 180 deg; joints [-28.091, 54.441, -85.065, 31.809, 116.704, 15.575]
  Call Extruder(205.69706)
  MoveL 7379 to (238.12, 41.97, 106.87) mm, rotated rx -180 ry 0 rz 180 deg; joints [-28.249, 54.496, -85.062, 31.964, 116.614, 15.617]
  MoveL 7380 to (238.12, 41.97, 106.87) mm, rotated rx -180 ry 0 rz 180 deg; joints [-28.249, 54.496, -85.062, 31.964, 116.614, 15.617]
  Call Extruder(205.81476)
  MoveL 7381 to (238.22, 42.15, 106.87) mm, rotated rx 180 ry 0 rz -180 deg; joints [-28.315, 54.514, -85.061, 32.031, 116.579, 15.638]
  MoveL 7382 to (238.22, 42.15, 106.87) mm, rotated rx 180 ry 0 rz -180 deg; joints [-28.315, 54.514, -85.061, 32.031, 116.579, 15.638]
  Call Extruder(206.02249)
  MoveL 7383 to (238.4, 42.45, 106.87) mm, rotated rx 180 ry 0 rz 180 deg; joints [-28.434, 54.546, -85.06, 32.149, 116.519, 15.675]
  MoveL 7384 to (238.4, 42.45, 106.87) mm, rotated rx 180 ry 0 rz 180 deg; joints [-28.434, 54.546, -85.06, 32.149, 116.519, 15.675]
  Call Extruder(206.22943)
  MoveL 7385 to (238.57, 42.75, 106.87) mm, rotated rx 180 ry 0 rz 180 deg; joints [-28.552, 54.579, -85.058, 32.267, 116.458, 15.711]
  MoveL 7386 to (238.57, 42.75, 106.87) mm, rotated rx 180 ry 0 rz 180 deg; joints [-28.552, 54.579, -85.058, 32.267, 116.458, 15.711]
  Call Extruder(206.43560)
  MoveL 7387 to (238.75, 43.06, 106.87) mm, rotated rx 180 ry 0 rz 180 deg; joints [-28.669, 54.611, -85.056, 32.384, 116.398, 15.747]
  MoveL 7388 to (238.75, 43.06, 106.87) mm, rotated rx 180 ry 0 rz 180 deg; joints [-28.669, 54.611, -85.056, 32.384, 116.398, 15.747]
  Call Extruder(206.61728)
  MoveL 7389 to (238.89, 43.34, 106.87) mm, rotated rx -180 ry 0 rz 180 deg; joints [-28.78, 54.639, -85.055, 32.496, 116.343, 15.783]
  MoveL 7390 to (238.89, 43.34, 106.87) mm, rotated rx -180 ry 0 rz 180 deg; joints [-28.78, 54.639, -85.055, 32.496, 116.343, 15.783]
  Call Extruder(206.77529)
  MoveL 7391 to (239, 43.58, 106.87) mm, rotated rx -180 ry 0 rz 180 deg; joints [-28.886, 54.662, -85.054, 32.603, 116.293, 15.819]
  MoveL 7392 to (239, 43.58, 106.87) mm, rotated rx -180 ry 0 rz 180 deg; joints [-28.886, 54.662, -85.054, 32.603, 116.293, 15.819]
  Call Extruder(206.93270)
  MoveL 7393 to (239.11, 43.83, 106.87) mm, rotated rx -180 ry 0 rz -180 deg; joints [-28.991, 54.685, -85.053, 32.71, 116.244, 15.854]
  MoveL 7394 to (239.11, 43.83, 106.87) mm, rotated rx -180 ry 0 rz -180 deg; joints [-28.991, 54.685, -85.053, 32.71, 116.244, 15.854]
  Call Extruder(207.11542)
  MoveL 7395 to (239.23, 44.13, 106.87) mm, rotated rx 180 ry 0 rz 180 deg; joints [-29.116, 54.712, -85.051, 32.836, 116.186, 15.896]
  MoveL 7396 to (239.23, 44.13, 106.87) mm, rotated rx 180 ry 0 rz 180 deg; joints [-29.116, 54.712, -85.051, 32.836, 116.186, 15.896]
  Call Extruder(207.29737)
  MoveL 7397 to (239.35, 44.42, 106.87) mm, rotated rx -180 ry 0 rz 180 deg; joints [-29.24, 54.738, -85.05, 32.961, 116.129, 15.937]
